C05459=1072.234,347.946,400.424,175.055,31.365,155.656
C05460=1072.241,348.193,400.389,175.059,31.371,155.657
C05461=1072.247,348.441,400.353,175.062,31.376,155.658
C05462=1072.254,348.688,400.318,175.066,31.382,155.659
C05463=1072.260,348.935,400.281,175.070,31.387,155.660
C05464=1072.266,349.183,400.246,175.073,31.392,155.661
C05465=1072.273,349.430,400.210,175.076,31.398,155.663
C05466=1072.279,349.678,400.175,175.080,31.403,155.664
C05467=1072.285,349.925,400.138,175.084,31.409,155.665
C05468=1072.292,350.172,400.103,175.087,31.415,155.666
C05469=1072.298,350.420,400.067,175.091,31.420,155.667
C05470=1072.304,350.667,400.031,175.095,31.426,155.668
C05471=1072.311,350.914,399.996,175.098,31.431,155.669
C05472=1072.317,351.162,399.960,175.101,31.436,155.670
C05473=1072.323,351.409,399.924,175.105,31.442,155.671
C05474=1072.330,351.656,399.889,175.109,31.448,155.672
C05475=1072.336,351.904,399.852,175.112,31.453,155.673
C05476=1072.342,352.151,399.816,175.116,31.458,155.674
C05477=1072.349,352.398,399.780,175.120,31.464,155.675
C05478=1072.356,352.646,399.745,175.123,31.470,155.676
C05479=1072.362,352.893,399.708,175.127,31.475,155.677
C05480=1072.368,353.140,399.673,175.131,31.481,155.679
C05481=1072.374,353.387,399.636,175.134,31.487,155.680
C05482=1072.380,353.635,399.600,175.137,31.492,155.681
C05483=1072.387,353.882,399.564,175.141,31.498,155.682
C05484=1072.393,354.129,399.528,175.145,31.503,155.683
C05485=1072.399,354.377,399.492,175.148,31.509,155.684
C05486=1072.406,354.624,399.456,175.152,31.515,155.685
C05487=1072.412,354.871,399.420,175.156,31.521,155.686
C05488=1072.418,355.118,399.384,175.160,31.526,155.687
C05489=1072.425,355.366,399.347,175.163,31.532,155.689
C05490=1072.432,355.613,399.311,175.167,31.537,155.690
C05491=1072.438,355.860,399.274,175.171,31.543,155.691
C05492=1072.444,356.108,399.238,175.174,31.549,155.692
C05493=1072.450,356.355,399.202,175.178,31.555,155.693
C05494=1072.457,356.602,399.165,175.182,31.561,155.694
C05495=1072.463,356.849,399.129,175.186,31.566,155.695
C05496=1072.470,357.097,399.092,175.189,31.572,155.696
C05497=1072.476,357.344,399.056,175.193,31.578,155.698
C05498=1072.482,357.592,399.020,175.197,31.583,155.699
C05499=1072.488,357.812,398.987,175.199,31.588,155.700
C05500=1072.495,358.032,398.955,175.203,31.594,155.701
C05501=1072.500,358.253,398.923,175.206,31.599,155.702
C05502=1072.506,358.474,398.889,175.210,31.604,155.703
C05503=1072.511,358.695,398.857,175.213,31.609,155.704
C05504=1072.517,358.916,398.824,175.216,31.615,155.705
C05505=1072.524,359.136,398.792,175.220,31.619,155.706
C05506=1072.529,359.357,398.759,175.223,31.625,155.707
C05507=1072.536,359.603,398.722,175.227,31.631,155.708
C05508=1072.542,359.851,398.685,175.230,31.637,155.709
C05509=1072.548,360.098,398.648,175.234,31.642,155.710
C05510=1072.554,360.346,398.612,175.238,31.648,155.711
C05511=1072.561,360.593,398.576,175.241,31.654,155.713
C05512=1072.568,360.840,398.539,175.245,31.660,155.714
C05513=1072.574,361.087,398.502,175.249,31.666,155.715
C05514=1072.580,361.334,398.465,175.253,31.672,155.716
C05515=1072.587,361.582,398.428,175.256,31.678,155.717
C05516=1072.593,361.829,398.391,175.260,31.684,155.719
C05517=1072.600,362.075,398.354,175.264,31.690,155.720
C05518=1072.607,362.323,398.317,175.269,31.696,155.721
C05519=1072.613,362.570,398.281,175.272,31.702,155.722
C05520=1072.619,362.817,398.243,175.276,31.708,155.723
C05521=1072.626,363.065,398.206,175.280,31.714,155.724
C05522=1072.632,363.312,398.170,175.284,31.720,155.726
C05523=1072.639,363.558,398.133,175.287,31.726,155.727
C05524=1072.645,363.806,398.095,175.291,31.732,155.728
C05525=1072.652,364.053,398.058,175.295,31.738,155.729
C05526=1072.659,364.300,398.021,175.299,31.744,155.730
C05527=1072.665,364.547,397.984,175.302,31.750,155.732
C05528=1072.671,364.794,397.947,175.306,31.756,155.733
C05529=1072.678,365.041,397.910,175.310,31.762,155.734
C05530=1072.684,365.289,397.873,175.314,31.769,155.735
C05531=1072.691,365.536,397.835,175.318,31.775,155.737
C05532=1072.697,365.783,397.797,175.322,31.781,155.738
C05533=1072.703,366.030,397.761,175.326,31.788,155.739
C05534=1072.710,366.277,397.723,175.330,31.793,155.740
C05535=1072.717,366.524,397.686,175.333,31.800,155.742
C05536=1072.723,366.771,397.649,175.337,31.806,155.743
C05537=1072.729,367.018,397.611,175.341,31.812,155.744
C05538=1072.736,367.265,397.573,175.345,31.819,155.745
C05539=1072.743,367.512,397.536,175.348,31.824,155.747
C05540=1072.749,367.760,397.498,175.353,31.831,155.748
C05541=1072.755,368.006,397.461,175.357,31.837,155.749
C05542=1072.762,368.254,397.423,175.361,31.844,155.751
C05543=1072.768,368.500,397.386,175.364,31.850,155.752
C05544=1072.775,368.748,397.348,175.368,31.856,155.753
C05545=1072.782,368.994,397.311,175.372,31.862,155.754
C05546=1072.788,369.242,397.272,175.376,31.869,155.756
C05547=1072.794,369.489,397.236,175.380,31.875,155.757
C05548=1072.801,369.736,397.198,175.384,31.882,155.758
C05549=1072.808,369.983,397.161,175.388,31.888,155.759
C05550=1072.814,370.230,397.123,175.392,31.894,155.761
C05551=1072.821,370.477,397.085,175.396,31.900,155.762
C05552=1072.828,370.723,397.047,175.399,31.907,155.763
C05553=1072.834,370.971,397.008,175.404,31.913,155.765
C05554=1072.841,371.217,396.971,175.408,31.920,155.766
C05555=1072.847,371.447,396.936,175.412,31.926,155.767
C05556=1072.854,371.676,396.901,175.415,31.932,155.768
C05557=1072.859,371.904,396.866,175.418,31.938,155.770
C05558=1072.865,372.134,396.830,175.422,31.944,155.771
C05559=1072.872,372.363,396.796,175.426,31.950,155.772
C05560=1072.878,372.592,396.761,175.430,31.956,155.773
C05561=1072.884,372.821,396.725,175.433,31.962,155.774
C05562=1072.890,373.051,396.690,175.437,31.968,155.776
C05563=1072.897,373.297,396.653,175.441,31.974,155.777
C05564=1072.904,373.544,396.614,175.445,31.981,155.778
C05565=1072.910,373.792,396.576,175.450,31.988,155.780
C05566=1072.916,374.038,396.538,175.453,31.994,155.781
C05567=1072.923,374.285,396.499,175.457,32.001,155.782
C05568=1072.929,374.533,396.461,175.461,32.007,155.784
C05569=1072.936,374.778,396.423,175.466,32.014,155.785
C05570=1072.943,375.026,396.385,175.470,32.021,155.787
C05571=1072.950,375.273,396.346,175.473,32.028,155.788
C05572=1072.956,375.520,396.308,175.477,32.034,155.789
C05573=1072.962,375.766,396.269,175.482,32.041,155.791
C05574=1072.969,376.014,396.231,175.486,32.048,155.792
C05575=1072.976,376.260,396.192,175.490,32.054,155.793
C05576=1072.982,376.508,396.154,175.493,32.061,155.795
C05577=1072.988,376.754,396.116,175.498,32.068,155.796
C05578=1072.995,377.001,396.077,175.502,32.075,155.798
C05579=1073.002,377.248,396.040,175.506,32.082,155.799
C05580=1073.009,377.495,396.001,175.511,32.089,155.801
C05581=1073.016,377.742,395.962,175.514,32.095,155.802
C05582=1073.023,377.989,395.924,175.518,32.102,155.803
C05583=1073.029,378.235,395.885,175.523,32.109,155.805
C05584=1073.036,378.482,395.846,175.527,32.116,155.806
C05585=1073.042,378.729,395.808,175.531,32.123,155.808
C05586=1073.049,378.976,395.769,175.534,32.129,155.809
C05587=1073.056,379.223,395.731,175.539,32.136,155.810
C05588=1073.062,379.470,395.692,175.543,32.143,155.812
C05589=1073.069,379.717,395.653,175.547,32.150,155.813
C05590=1073.076,379.964,395.614,175.552,32.157,155.815
C05591=1073.083,380.210,395.575,175.556,32.164,155.816
C05592=1073.090,380.457,395.536,175.560,32.171,155.818
C05593=1073.096,380.703,395.498,175.564,32.178,155.819
C05594=1073.103,380.951,395.459,175.568,32.185,155.820
C05595=1073.110,381.197,395.420,175.573,32.192,155.822
C05596=1073.117,381.445,395.381,175.577,32.199,155.823
C05597=1073.124,381.691,395.342,175.581,32.206,155.825
C05598=1073.131,381.938,395.303,175.585,32.213,155.826
C05599=1073.136,382.185,395.264,175.589,32.220,155.828
C05600=1073.143,382.431,395.225,175.594,32.227,155.829
C05601=1073.150,382.678,395.186,175.598,32.235,155.831
C05602=1073.157,382.924,395.147,175.602,32.241,155.832
C05603=1073.163,383.172,395.108,175.607,32.249,155.834
C05604=1073.170,383.418,395.069,175.610,32.256,155.835
C05605=1073.177,383.665,395.029,175.614,32.263,155.837
C05606=1073.183,383.912,394.990,175.619,32.271,155.838
C05607=1073.190,384.159,394.951,175.623,32.278,155.840
C05608=1073.197,384.405,394.911,175.628,32.285,155.841
C05609=1073.204,384.652,394.873,175.632,32.292,155.843
C05610=1073.211,384.899,394.832,175.637,32.300,155.845
C05611=1073.217,385.142,394.794,175.640,32.307,155.846
C05612=1073.224,385.386,394.755,175.644,32.314,155.848
C05613=1073.231,385.630,394.716,175.649,32.321,155.849
C05614=1073.237,385.873,394.677,175.653,32.328,155.851
C05615=1073.244,386.117,394.638,175.658,32.336,155.852
C05616=1073.250,386.361,394.599,175.662,32.343,155.854
C05617=1073.257,386.605,394.560,175.666,32.350,155.855
C05618=1073.264,386.848,394.521,175.670,32.358,155.857
C05619=1073.270,387.096,394.481,175.674,32.365,155.858
C05620=1073.278,387.342,394.442,175.679,32.373,155.860
C05621=1073.285,387.588,394.402,175.683,32.380,155.862
C05622=1073.291,387.836,394.362,175.688,32.388,155.863
C05623=1073.299,388.082,394.323,175.692,32.395,155.865
C05624=1073.305,388.328,394.283,175.697,32.402,155.866
C05625=1073.312,388.575,394.244,175.701,32.410,155.868
C05626=1073.319,388.822,394.204,175.706,32.418,155.870
C05627=1073.326,389.069,394.164,175.709,32.425,155.871
C05628=1073.333,389.315,394.124,175.714,32.432,155.873
C05629=1073.339,389.561,394.084,175.718,32.440,155.874
C05630=1073.347,389.808,394.044,175.723,32.448,155.876
C05631=1073.354,390.055,394.005,175.728,32.456,155.878
C05632=1073.361,390.301,393.964,175.732,32.463,155.879
C05633=1073.368,390.549,393.925,175.737,32.471,155.881
C05634=1073.374,390.795,393.885,175.741,32.478,155.882
C05635=1073.382,391.042,393.845,175.746,32.486,155.884
C05636=1073.388,391.289,393.805,175.749,32.494,155.886
C05637=1073.396,391.534,393.765,175.754,32.502,155.887
C05638=1073.403,391.781,393.724,175.759,32.509,155.889
C05639=1073.409,392.028,393.684,175.763,32.517,155.891
C05640=1073.416,392.274,393.645,175.768,32.525,155.893
C05641=1073.423,392.521,393.604,175.772,32.533,155.894
C05642=1073.430,392.768,393.564,175.777,32.541,155.896
C05643=1073.437,393.013,393.524,175.782,32.548,155.897
C05644=1073.444,393.261,393.483,175.786,32.556,155.899
C05645=1073.450,393.507,393.443,175.791,32.564,155.901
C05646=1073.457,393.754,393.402,175.795,32.573,155.903
C05647=1073.465,394.000,393.362,175.800,32.580,155.904
C05648=1073.472,394.247,393.322,175.805,32.588,155.906
C05649=1073.478,394.494,393.282,175.808,32.596,155.908
C05650=1073.486,394.740,393.240,175.813,32.604,155.909
C05651=1073.492,394.987,393.200,175.818,32.613,155.911
C05652=1073.500,395.233,393.160,175.822,32.620,155.913
C05653=1073.506,395.480,393.119,175.827,32.628,155.915
C05654=1073.514,395.726,393.078,175.832,32.637,155.917
C05655=1073.520,395.973,393.038,175.836,32.645,155.918
C05656=1073.527,396.219,392.997,175.841,32.653,155.920
C05657=1073.534,396.466,392.957,175.846,32.661,155.922
C05658=1073.541,396.712,392.915,175.850,32.669,155.924
C05659=1073.548,396.959,392.874,175.855,32.678,155.925
C05660=1073.555,397.205,392.835,175.860,32.686,155.927
C05661=1073.563,397.452,392.793,175.864,32.694,155.929
C05662=1073.570,397.698,392.752,175.869,32.702,155.931
C05663=1073.576,397.945,392.712,175.874,32.711,155.933
C05664=1073.584,398.191,392.671,175.878,32.718,155.934
C05665=1073.591,398.438,392.630,175.883,32.727,155.936
C05666=1073.598,398.684,392.589,175.888,32.735,155.938
C05667=1073.605,398.941,392.546,175.893,32.744,155.940
C05668=1073.612,399.197,392.503,175.898,32.753,155.942
C05669=1073.620,399.453,392.460,175.903,32.762,155.944
C05670=1073.627,399.709,392.418,175.908,32.771,155.946
C05671=1073.634,399.956,392.376,175.912,32.779,155.948
C05672=1073.641,400.202,392.335,175.917,32.787,155.949
C05673=1073.648,400.448,392.294,175.922,32.796,155.951
C05674=1073.655,400.695,392.253,175.927,32.805,155.953
C05675=1073.663,400.942,392.212,175.931,32.813,155.955
C05676=1073.669,401.188,392.170,175.936,32.822,155.957
C05677=1073.676,401.434,392.129,175.941,32.830,155.959
C05678=1073.683,401.681,392.088,175.946,32.839,155.961
C05679=1073.690,401.928,392.047,175.951,32.847,155.963
C05680=1073.698,402.174,392.005,175.955,32.856,155.965
C05681=1073.705,402.421,391.964,175.960,32.865,155.966
C05682=1073.712,402.667,391.922,175.965,32.873,155.968
C05683=1073.719,402.914,391.880,175.970,32.882,155.970
C05684=1073.726,403.160,391.839,175.975,32.891,155.972
C05685=1073.733,403.405,391.798,175.980,32.900,155.974
C05686=1073.741,403.652,391.756,175.985,32.909,155.976
C05687=1073.747,403.899,391.715,175.989,32.917,155.978
C05688=1073.755,404.145,391.673,175.994,32.926,155.980
C05689=1073.762,404.392,391.631,175.999,32.935,155.982
C05690=1073.769,404.638,391.589,176.004,32.944,155.984
C05691=1073.776,404.884,391.548,176.009,32.953,155.986
C05692=1073.784,405.130,391.506,176.014,32.962,155.988
C05693=1073.790,405.377,391.464,176.019,32.971,155.990
C05694=1073.798,405.623,391.422,176.024,32.980,155.992
C05695=1073.805,405.870,391.380,176.030,32.989,155.994
C05696=1073.812,406.116,391.338,176.035,32.998,155.996
C05697=1073.819,406.362,391.296,176.039,33.007,155.998
C05698=1073.826,406.609,391.254,176.044,33.016,156.000
C05699=1073.834,406.855,391.212,176.049,33.026,156.002
C05700=1073.841,407.101,391.170,176.054,33.035,156.004
C05701=1073.848,407.348,391.127,176.059,33.044,156.006
C05702=1073.855,407.595,391.086,176.064,33.053,156.008
C05703=1073.862,407.841,391.043,176.069,33.063,156.010
C05704=1073.870,408.087,391.001,176.074,33.072,156.012
C05705=1073.877,408.333,390.959,176.079,33.081,156.015
C05706=1073.884,408.580,390.916,176.085,33.090,156.017
C05707=1073.891,408.826,390.874,176.090,33.100,156.019
C05708=1073.898,409.072,390.832,176.095,33.109,156.021
C05709=1073.906,409.319,390.789,176.100,33.119,156.023
C05710=1073.913,409.565,390.747,176.105,33.128,156.025
C05711=1073.920,409.811,390.704,176.110,33.137,156.027
C05712=1073.928,410.057,390.662,176.116,33.147,156.029
C05713=1073.934,410.303,390.620,176.121,33.157,156.031
C05714=1073.942,410.550,390.577,176.127,33.166,156.034
C05715=1073.950,410.796,390.534,176.132,33.175,156.036
C05716=1073.957,411.042,390.492,176.137,33.185,156.038
C05717=1073.963,411.288,390.449,176.142,33.195,156.040
C05718=1073.972,411.535,390.407,176.147,33.204,156.042
C05719=1073.979,411.781,390.364,176.152,33.214,156.044
C05720=1073.986,412.027,390.321,176.158,33.224,156.047
C05721=1073.993,412.274,390.278,176.164,33.233,156.049
C05722=1074.001,412.519,390.236,176.169,33.243,156.051
C05723=1074.009,412.779,390.190,176.174,33.254,156.053
C05724=1074.017,413.038,390.145,176.180,33.264,156.056
C05725=1074.024,413.298,390.100,176.186,33.274,156.058
C05726=1074.032,413.558,390.055,176.192,33.284,156.060
C05727=1074.040,413.804,390.012,176.197,33.294,156.063
C05728=1074.047,414.050,389.968,176.202,33.304,156.065
C05729=1074.055,414.297,389.925,176.207,33.314,156.067
C05730=1074.063,414.542,389.883,176.213,33.324,156.069
C05731=1074.070,414.789,389.840,176.219,33.334,156.072
C05732=1074.077,415.035,389.797,176.224,33.344,156.074
C05733=1074.085,415.281,389.753,176.229,33.354,156.076
C05734=1074.092,415.527,389.710,176.235,33.364,156.078
C05735=1074.100,415.774,389.667,176.241,33.374,156.081
C05736=1074.107,416.019,389.624,176.246,33.385,156.083
C05737=1074.115,416.266,389.580,176.251,33.395,156.086
C05738=1074.122,416.512,389.537,176.257,33.405,156.088
C05739=1074.129,416.758,389.493,176.263,33.415,156.090
C05740=1074.137,417.004,389.450,176.268,33.425,156.093
C05741=1074.144,417.250,389.406,176.274,33.436,156.095
C05742=1074.152,417.496,389.363,176.280,33.446,156.097
C05743=1074.159,417.742,389.319,176.285,33.456,156.100
C05744=1074.167,417.988,389.276,176.291,33.467,156.102
C05745=1074.174,418.234,389.232,176.296,33.477,156.105
C05746=1074.182,418.480,389.188,176.302,33.488,156.107
C05747=1074.189,418.726,389.144,176.308,33.499,156.109
C05748=1074.197,418.972,389.101,176.313,33.509,156.112
C05749=1074.204,419.218,389.057,176.320,33.519,156.114
C05750=1074.212,419.464,389.013,176.325,33.530,156.117
C05751=1074.220,419.711,388.969,176.330,33.541,156.119
C05752=1074.227,419.956,388.926,176.337,33.551,156.121
C05753=1074.235,420.202,388.881,176.342,33.562,156.124
C05754=1074.243,420.448,388.838,176.348,33.573,156.126
C05755=1074.250,420.694,388.793,176.354,33.583,156.129
C05756=1074.258,420.941,388.749,176.360,33.594,156.131
C05757=1074.266,421.186,388.705,176.365,33.605,156.134
C05758=1074.273,421.432,388.662,176.372,33.615,156.136
C05759=1074.282,421.678,388.617,176.377,33.627,156.139
C05760=1074.289,421.924,388.572,176.383,33.638,156.142
C05761=1074.297,422.170,388.529,176.389,33.648,156.144
C05762=1074.303,422.416,388.484,176.395,33.660,156.147
C05763=1074.311,422.661,388.440,176.401,33.670,156.149
C05764=1074.319,422.907,388.396,176.407,33.682,156.152
C05765=1074.327,423.154,388.351,176.413,33.692,156.154
C05766=1074.335,423.400,388.307,176.419,33.704,156.157
C05767=1074.342,423.646,388.262,176.425,33.715,156.160
C05768=1074.350,423.891,388.218,176.431,33.726,156.162
C05769=1074.358,424.137,388.173,176.437,33.737,156.165
C05770=1074.365,424.383,388.128,176.444,33.748,156.167
C05771=1074.373,424.629,388.084,176.449,33.760,156.170
C05772=1074.381,424.875,388.039,176.456,33.771,156.173
C05773=1074.389,425.121,387.995,176.461,33.783,156.175
C05774=1074.396,425.367,387.950,176.467,33.794,156.178
C05775=1074.405,425.612,387.905,176.474,33.805,156.181
C05776=1074.412,425.858,387.860,176.480,33.817,156.184
C05777=1074.420,426.104,387.816,176.486,33.828,156.186
C05778=1074.427,426.350,387.771,176.492,33.839,156.189
C05779=1074.437,426.627,387.720,176.499,33.853,156.192
C05780=1074.446,426.905,387.669,176.507,33.866,156.195
C05781=1074.455,427.182,387.618,176.513,33.879,156.198
C05782=1074.464,427.459,387.568,176.521,33.892,156.201
C05783=1074.471,427.705,387.523,176.527,33.904,156.204
C05784=1074.479,427.951,387.477,176.533,33.915,156.207
C05785=1074.487,428.197,387.433,176.539,33.928,156.210
C05786=1074.495,428.443,387.387,176.546,33.939,156.212
C05787=1074.503,428.688,387.341,176.552,33.951,156.215
C05788=1074.510,428.934,387.296,176.559,33.963,156.218
C05789=1074.518,429.179,387.251,176.565,33.975,156.221
C05790=1074.527,429.425,387.205,176.571,33.987,156.224
C05791=1074.534,429.671,387.160,176.578,33.999,156.227
C05792=1074.542,429.917,387.115,176.584,34.011,156.230
C05793=1074.551,430.163,387.069,176.591,34.023,156.232
C05794=1074.558,430.408,387.024,176.598,34.035,156.235
C05795=1074.566,430.654,386.978,176.604,34.047,156.238
C05796=1074.574,430.900,386.932,176.611,34.060,156.241
C05797=1074.582,431.145,386.887,176.618,34.072,156.244
C05798=1074.590,431.390,386.841,176.624,34.084,156.247
C05799=1074.598,431.636,386.795,176.630,34.097,156.250
C05800=1074.606,431.882,386.750,176.637,34.109,156.253
C05801=1074.614,432.128,386.704,176.643,34.121,156.256
C05802=1074.622,432.373,386.657,176.650,34.134,156.259
C05803=1074.630,432.619,386.611,176.657,34.146,156.262
C05804=1074.638,432.864,386.566,176.663,34.159,156.265
C05805=1074.646,433.109,386.519,176.670,34.171,156.268
C05806=1074.654,433.355,386.473,176.677,34.184,156.271
C05807=1074.662,433.601,386.428,176.684,34.197,156.274
C05808=1074.670,433.846,386.381,176.690,34.209,156.277
C05809=1074.678,434.092,386.335,176.698,34.223,156.280
C05810=1074.687,434.337,386.289,176.705,34.235,156.283
C05811=1074.694,434.583,386.243,176.712,34.248,156.286
C05812=1074.703,434.828,386.196,176.719,34.261,156.290
C05813=1074.711,435.074,386.149,176.725,34.274,156.293
C05814=1074.719,435.319,386.104,176.732,34.287,156.296
C05815=1074.728,435.565,386.057,176.739,34.300,156.299
C05816=1074.735,435.809,386.011,176.746,34.313,156.302
C05817=1074.743,436.055,385.963,176.754,34.326,156.305
C05818=1074.752,436.301,385.917,176.760,34.339,156.308
C05819=1074.760,436.547,385.871,176.767,34.352,156.312
C05820=1074.768,436.792,385.824,176.774,34.365,156.315
C05821=1074.777,437.037,385.778,176.781,34.378,156.318
C05822=1074.785,437.283,385.731,176.789,34.392,156.321
C05823=1074.794,437.528,385.684,176.796,34.405,156.325
C05824=1074.802,437.773,385.638,176.803,34.418,156.328
C05825=1074.809,438.019,385.590,176.810,34.432,156.331
C05826=1074.818,438.264,385.544,176.818,34.445,156.334
C05827=1074.827,438.509,385.496,176.825,34.459,156.338
C05828=1074.835,438.755,385.449,176.831,34.472,156.341
C05829=1074.844,439.000,385.403,176.839,34.486,156.344
C05830=1074.852,439.246,385.355,176.846,34.499,156.348
C05831=1074.861,439.491,385.308,176.853,34.513,156.351
C05832=1074.869,439.737,385.261,176.861,34.527,156.354
C05833=1074.877,439.981,385.214,176.868,34.541,156.358
C05834=1074.885,440.227,385.167,176.875,34.555,156.361
C05835=1074.895,440.518,385.110,176.885,34.571,156.365
C05836=1074.906,440.809,385.054,176.894,34.588,156.369
C05837=1074.916,441.103,384.997,176.902,34.604,156.374
C05838=1074.926,441.397,384.941,176.911,34.621,156.378
C05839=1074.935,441.690,384.883,176.921,34.638,156.382
C05840=1074.946,441.985,384.826,176.930,34.655,156.386
C05841=1074.954,442.230,384.778,176.937,34.670,156.390
C05842=1074.963,442.475,384.731,176.945,34.684,156.393
C05843=1074.971,442.720,384.683,176.953,34.698,156.397
C05844=1074.980,442.965,384.635,176.961,34.713,156.400
C05845=1074.988,443.211,384.587,176.968,34.727,156.404
C05846=1074.997,443.456,384.539,176.976,34.742,156.408
C05847=1075.006,443.701,384.491,176.984,34.756,156.411
C05848=1075.014,443.946,384.444,176.992,34.771,156.415
C05849=1075.023,444.191,384.395,177.000,34.785,156.418
C05850=1075.032,444.437,384.347,177.007,34.800,156.422
C05851=1075.040,444.682,384.299,177.015,34.815,156.426
C05852=1075.048,444.927,384.251,177.024,34.829,156.429
C05853=1075.057,445.171,384.202,177.031,34.844,156.433
C05854=1075.066,445.417,384.154,177.039,34.859,156.437
C05855=1075.075,445.662,384.106,177.047,34.874,156.441
C05856=1075.083,445.907,384.058,177.056,34.889,156.445
C05857=1075.092,446.152,384.009,177.063,34.904,156.448
C05858=1075.101,446.396,383.961,177.072,34.919,156.452
C05859=1075.110,446.642,383.912,177.080,34.935,156.456
C05860=1075.118,446.887,383.863,177.088,34.950,156.460
C05861=1075.127,447.131,383.815,177.096,34.965,156.464
C05862=1075.136,447.377,383.765,177.103,34.980,156.467
C05863=1075.145,447.622,383.718,177.111,34.995,156.471
C05864=1075.154,447.867,383.669,177.118,35.010,156.475
C05865=1075.162,448.111,383.620,177.124,35.026,156.479
C05866=1075.171,448.355,383.571,177.131,35.041,156.483
C05867=1075.180,448.600,383.523,177.137,35.056,156.487
C05868=1075.190,448.845,383.474,177.144,35.071,156.491
C05869=1075.201,449.089,383.427,177.149,35.085,156.494
C05870=1075.213,449.334,383.380,177.155,35.099,156.498
C05871=1075.226,449.579,383.334,177.161,35.112,156.501
C05872=1075.242,449.825,383.289,177.166,35.124,156.504
C05873=1074.885,449.822,383.050,177.148,35.277,156.545
C05874=1074.870,449.576,383.095,177.141,35.264,156.542
C05875=1074.856,449.331,383.142,177.136,35.251,156.538
C05876=1074.844,449.085,383.188,177.130,35.238,156.535
C05877=1074.832,448.841,383.235,177.124,35.223,156.531
C05878=1074.823,448.596,383.284,177.117,35.209,156.527
C05879=1074.814,448.352,383.333,177.111,35.193,156.523
C05880=1074.805,448.108,383.381,177.104,35.178,156.519
C05881=1074.796,447.863,383.430,177.098,35.163,156.516
C05882=1074.787,447.619,383.478,177.090,35.148,156.512
C05883=1074.778,447.374,383.527,177.083,35.133,156.508
C05884=1074.769,447.129,383.577,177.075,35.118,156.504
C05885=1074.761,446.884,383.625,177.067,35.102,156.500
C05886=1074.752,446.639,383.674,177.059,35.088,156.496
C05887=1074.742,446.394,383.723,177.051,35.072,156.492
C05888=1074.734,446.149,383.771,177.042,35.057,156.489
C05889=1074.725,445.904,383.820,177.034,35.042,156.485
C05890=1074.717,445.659,383.869,177.025,35.027,156.481
C05891=1074.707,445.414,383.916,177.018,35.012,156.477
C05892=1074.699,445.169,383.965,177.010,34.997,156.474
C05893=1074.691,444.924,384.013,177.001,34.982,156.470
C05894=1074.681,444.679,384.062,176.994,34.968,156.466
C05895=1074.673,444.434,384.110,176.985,34.953,156.462
C05896=1074.665,444.189,384.158,176.977,34.938,156.459
C05897=1074.655,443.944,384.206,176.970,34.924,156.455
C05898=1074.647,443.698,384.254,176.962,34.909,156.451
C05899=1074.639,443.453,384.302,176.953,34.895,156.448
C05900=1074.630,443.208,384.350,176.946,34.880,156.444
C05901=1074.622,442.963,384.398,176.938,34.866,156.441
C05902=1074.613,442.717,384.446,176.930,34.851,156.437
C05903=1074.604,442.472,384.494,176.922,34.837,156.433
C05904=1074.596,442.227,384.541,176.915,34.823,156.430
C05905=1074.587,441.982,384.589,176.907,34.808,156.426
C05906=1074.579,441.772,384.631,176.901,34.796,156.423
C05907=1074.573,441.561,384.671,176.894,34.784,156.420
C05908=1074.565,441.349,384.713,176.887,34.772,156.417
C05909=1074.558,441.139,384.753,176.881,34.760,156.414
C05910=1074.551,440.927,384.794,176.874,34.748,156.411
C05911=1074.543,440.717,384.835,176.868,34.736,156.408
C05912=1074.536,440.506,384.877,176.861,34.724,156.405
C05913=1074.529,440.295,384.917,176.855,34.712,156.402
C05914=1074.520,440.050,384.964,176.847,34.698,156.399
C05915=1074.512,439.805,385.012,176.839,34.684,156.395
C05916=1074.503,439.559,385.058,176.832,34.670,156.392
C05917=1074.495,439.314,385.106,176.824,34.657,156.389
C05918=1074.487,439.068,385.153,176.817,34.643,156.385
C05919=1074.478,438.823,385.200,176.809,34.630,156.382
C05920=1074.469,438.578,385.247,176.802,34.616,156.379
C05921=1074.462,438.332,385.295,176.795,34.602,156.375
C05922=1074.453,438.087,385.341,176.788,34.589,156.372
C05923=1074.445,437.842,385.388,176.780,34.576,156.369
C05924=1074.436,437.597,385.435,176.773,34.562,156.365
C05925=1074.428,437.351,385.482,176.766,34.549,156.362
C05926=1074.419,437.106,385.529,176.758,34.536,156.359
C05927=1074.411,436.860,385.575,176.751,34.522,156.356
C05928=1074.403,436.615,385.622,176.744,34.509,156.352
C05929=1074.395,436.370,385.669,176.737,34.496,156.349
C05930=1074.386,436.124,385.716,176.730,34.483,156.346
C05931=1074.378,435.879,385.762,176.722,34.470,156.343
C05932=1074.370,435.633,385.808,176.716,34.457,156.340
C05933=1074.362,435.388,385.855,176.709,34.444,156.337
C05934=1074.353,435.142,385.902,176.702,34.431,156.333
C05935=1074.345,434.898,385.948,176.695,34.418,156.330
C05936=1074.337,434.651,385.994,176.688,34.405,156.327
C05937=1074.329,434.407,386.040,176.681,34.392,156.324
C05938=1074.320,434.161,386.087,176.674,34.380,156.321
C05939=1074.313,433.915,386.134,176.667,34.367,156.318
C05940=1074.305,433.670,386.180,176.660,34.354,156.315
C05941=1074.297,433.424,386.226,176.653,34.341,156.312
C05942=1074.289,433.179,386.272,176.646,34.328,156.309
C05943=1074.280,432.933,386.318,176.639,34.316,156.306
C05944=1074.273,432.687,386.364,176.632,34.304,156.303
C05945=1074.264,432.442,386.411,176.626,34.291,156.299
C05946=1074.257,432.196,386.456,176.619,34.278,156.296
C05947=1074.248,431.950,386.502,176.612,34.266,156.293
C05948=1074.241,431.705,386.548,176.605,34.253,156.290
C05949=1074.232,431.460,386.594,176.600,34.241,156.287
C05950=1074.223,431.192,386.644,176.592,34.228,156.284
C05951=1074.215,430.924,386.694,176.585,34.215,156.281
C05952=1074.206,430.656,386.743,176.577,34.201,156.278
C05953=1074.197,430.389,386.793,176.570,34.188,156.275
C05954=1074.189,430.142,386.839,176.564,34.176,156.272
C05955=1074.181,429.896,386.884,176.557,34.164,156.269
C05956=1074.174,429.651,386.930,176.550,34.151,156.266
C05957=1074.165,429.405,386.975,176.544,34.140,156.263
C05958=1074.157,429.160,387.021,176.537,34.128,156.260
C05959=1074.149,428.914,387.067,176.531,34.116,156.257
C05960=1074.141,428.668,387.113,176.525,34.104,156.255
C05961=1074.133,428.422,387.157,176.518,34.092,156.252
C05962=1074.125,428.177,387.203,176.511,34.080,156.249
C05963=1074.118,427.931,387.247,176.505,34.068,156.246
C05964=1074.110,427.686,387.293,176.499,34.057,156.243
C05965=1074.102,427.440,387.339,176.493,34.045,156.241
C05966=1074.093,427.183,387.386,176.486,34.033,156.238
C05967=1074.085,426.926,387.433,176.479,34.020,156.235
C05968=1074.077,426.669,387.480,176.473,34.009,156.232
C05969=1074.069,426.412,387.527,176.466,33.996,156.229
C05970=1074.061,426.166,387.571,176.460,33.985,156.226
C05971=1074.053,425.920,387.616,176.453,33.973,156.224
C05972=1074.045,425.675,387.661,176.447,33.962,156.221
C05973=1074.037,425.429,387.706,176.441,33.950,156.218
C05974=1074.029,425.183,387.750,176.434,33.939,156.216
C05975=1074.022,424.937,387.795,176.429,33.928,156.213
C05976=1074.014,424.692,387.840,176.422,33.917,156.210
C05977=1074.007,424.446,387.884,176.416,33.905,156.208
C05978=1073.998,424.200,387.930,176.410,33.894,156.205
C05979=1073.990,423.955,387.974,176.404,33.883,156.202
C05980=1073.983,423.709,388.019,176.398,33.872,156.200
C05981=1073.975,423.463,388.063,176.392,33.860,156.197
C05982=1073.968,423.216,388.107,176.385,33.850,156.195
C05983=1073.960,422.971,388.152,176.380,33.838,156.192
C05984=1073.952,422.724,388.197,176.373,33.827,156.189
C05985=1073.944,422.479,388.241,176.368,33.816,156.187
C05986=1073.936,422.233,388.285,176.361,33.805,156.184
C05987=1073.929,421.987,388.330,176.356,33.794,156.182
C05988=1073.921,421.741,388.374,176.349,33.783,156.179
C05989=1073.914,421.496,388.418,176.344,33.772,156.176
C05990=1073.906,421.249,388.463,176.338,33.761,156.174
C05991=1073.899,421.003,388.506,176.332,33.751,156.171
C05992=1073.891,420.757,388.551,176.326,33.740,156.169
C05993=1073.883,420.511,388.594,176.320,33.730,156.166
C05994=1073.875,420.265,388.639,176.314,33.719,156.164
C05995=1073.868,420.019,388.683,176.308,33.708,156.161
C05996=1073.860,419.774,388.727,176.302,33.697,156.159
C05997=1073.852,419.527,388.770,176.297,33.687,156.157
C05998=1073.845,419.281,388.814,176.290,33.676,156.154
C05999=1073.837,419.035,388.858,176.285,33.666,156.152
C06000=1073.829,418.789,388.902,176.280,33.655,156.149
C06001=1073.822,418.543,388.945,176.273,33.645,156.147
C06002=1073.814,418.297,388.989,176.268,33.634,156.144
C06003=1073.806,418.051,389.033,176.262,33.624,156.142
C06004=1073.799,417.805,389.077,176.256,33.613,156.140
C06005=1073.792,417.559,389.121,176.251,33.603,156.137
C06006=1073.785,417.313,389.164,176.244,33.593,156.135
C06007=1073.777,417.067,389.208,176.239,33.582,156.132
C06008=1073.769,416.820,389.251,176.234,33.572,156.130
C06009=1073.762,416.574,389.294,176.228,33.562,156.128
C06010=1073.754,416.328,389.338,176.222,33.551,156.125
C06011=1073.747,416.082,389.381,176.217,33.541,156.123
C06012=1073.739,415.836,389.425,176.212,33.531,156.121
C06013=1073.732,415.590,389.468,176.205,33.521,156.118
C06014=1073.724,415.344,389.512,176.200,33.511,156.116
C06015=1073.717,415.098,389.555,176.195,33.501,156.114
C06016=1073.710,414.851,389.598,176.189,33.491,156.111
C06017=1073.702,414.605,389.642,176.183,33.481,156.109
C06018=1073.694,414.360,389.684,176.178,33.471,156.107
C06019=1073.686,414.113,389.727,176.172,33.461,156.105
C06020=1073.679,413.867,389.770,176.167,33.451,156.102
C06021=1073.672,413.621,389.814,176.161,33.441,156.100
C06022=1073.663,413.360,389.859,176.156,33.431,156.098
C06023=1073.656,413.099,389.905,176.149,33.420,156.095
C06024=1073.648,412.838,389.949,176.144,33.410,156.093
C06025=1073.639,412.577,389.996,176.139,33.399,156.091
C06026=1073.632,412.330,390.039,176.133,33.390,156.088
C06027=1073.625,412.085,390.080,176.127,33.380,156.086
C06028=1073.617,411.838,390.124,176.122,33.370,156.084
C06029=1073.610,411.592,390.167,176.117,33.361,156.082
C06030=1073.603,411.346,390.210,176.112,33.351,156.080
C06031=1073.595,411.100,390.252,176.107,33.341,156.077
C06032=1073.588,410.853,390.295,176.101,33.332,156.075
C06033=1073.581,410.607,390.337,176.096,33.322,156.073
C06034=1073.573,410.361,390.380,176.090,33.313,156.071
C06035=1073.566,410.115,390.423,176.085,33.304,156.069
C06036=1073.559,409.868,390.465,176.080,33.294,156.067
C06037=1073.551,409.622,390.507,176.074,33.284,156.065
C06038=1073.544,409.375,390.550,176.069,33.275,156.062
C06039=1073.537,409.129,390.593,176.064,33.266,156.060
C06040=1073.529,408.883,390.635,176.059,33.256,156.058
C06041=1073.523,408.637,390.677,176.054,33.247,156.056
C06042=1073.515,408.391,390.719,176.048,33.238,156.054
C06043=1073.508,408.145,390.762,176.043,33.228,156.052
C06044=1073.501,407.898,390.805,176.038,33.219,156.050
C06045=1073.493,407.652,390.847,176.033,33.210,156.048
C06046=1073.486,407.405,390.889,176.028,33.200,156.046
C06047=1073.479,407.159,390.931,176.023,33.191,156.043
C06048=1073.472,406.913,390.974,176.018,33.182,156.042
C06049=1073.465,406.666,391.015,176.012,33.173,156.039
C06050=1073.458,406.420,391.057,176.007,33.164,156.037
C06051=1073.450,406.174,391.099,176.002,33.155,156.035
C06052=1073.443,405.928,391.142,175.998,33.146,156.033
C06053=1073.436,405.681,391.183,175.993,33.136,156.031
C06054=1073.429,405.435,391.226,175.988,33.128,156.029
C06055=1073.422,405.188,391.267,175.983,33.119,156.027
C06056=1073.414,404.942,391.309,175.977,33.109,156.025
C06057=1073.407,404.696,391.351,175.972,33.100,156.023
C06058=1073.400,404.450,391.393,175.967,33.092,156.021
C06059=1073.392,404.204,391.435,175.962,33.083,156.019
C06060=1073.386,403.957,391.476,175.957,33.074,156.017
C06061=1073.379,403.710,391.518,175.952,33.065,156.015
C06062=1073.371,403.464,391.560,175.948,33.056,156.013
C06063=1073.364,403.217,391.601,175.943,33.047,156.011
C06064=1073.357,402.971,391.643,175.938,33.038,156.009
C06065=1073.350,402.725,391.685,175.933,33.030,156.008
C06066=1073.342,402.478,391.726,175.928,33.021,156.006
C06067=1073.335,402.231,391.767,175.922,33.012,156.004
C06068=1073.328,401.985,391.810,175.918,33.004,156.002
C06069=1073.321,401.739,391.851,175.913,32.995,156.000
C06070=1073.314,401.492,391.892,175.908,32.987,155.998
C06071=1073.307,401.246,391.933,175.903,32.978,155.996
C06072=1073.300,401.000,391.974,175.898,32.970,155.994
C06073=1073.292,400.753,392.015,175.894,32.961,155.992
C06074=1073.285,400.506,392.057,175.889,32.952,155.990
C06075=1073.278,400.260,392.099,175.884,32.944,155.989
C06076=1073.271,400.013,392.140,175.879,32.935,155.987
C06077=1073.264,399.768,392.181,175.875,32.927,155.985
C06078=1073.256,399.510,392.224,175.870,32.918,155.983
C06079=1073.249,399.251,392.267,175.865,32.909,155.981
C06080=1073.242,398.994,392.310,175.860,32.901,155.979
C06081=1073.234,398.736,392.353,175.855,32.892,155.977
C06082=1073.228,398.490,392.394,175.850,32.883,155.975
C06083=1073.221,398.243,392.435,175.845,32.875,155.973
C06084=1073.214,397.996,392.476,175.841,32.867,155.972
C06085=1073.206,397.750,392.517,175.836,32.858,155.970
C06086=1073.200,397.504,392.558,175.831,32.850,155.968
C06087=1073.193,397.257,392.598,175.827,32.842,155.966
C06088=1073.185,397.010,392.640,175.822,32.834,155.964
C06089=1073.179,396.764,392.680,175.817,32.826,155.963
C06090=1073.171,396.517,392.720,175.813,32.817,155.961
C06091=1073.164,396.271,392.761,175.808,32.809,155.959
C06092=1073.157,396.025,392.802,175.803,32.801,155.957
C06093=1073.150,395.778,392.843,175.799,32.793,155.956
C06094=1073.143,395.532,392.884,175.794,32.785,155.954
C06095=1073.136,395.285,392.924,175.789,32.776,155.952
C06096=1073.130,395.039,392.965,175.785,32.769,155.950
C06097=1073.122,394.792,393.005,175.780,32.761,155.949
C06098=1073.115,394.546,393.046,175.775,32.752,155.947
C06099=1073.108,394.299,393.087,175.771,32.744,155.945
C06100=1073.101,394.053,393.127,175.766,32.736,155.943
C06101=1073.095,393.806,393.168,175.762,32.729,155.942
C06102=1073.087,393.559,393.207,175.757,32.721,155.940
C06103=1073.080,393.313,393.249,175.752,32.713,155.938
C06104=1073.074,393.066,393.289,175.748,32.705,155.937
C06105=1073.066,392.819,393.329,175.743,32.697,155.935
C06106=1073.060,392.573,393.369,175.739,32.689,155.933
C06107=1073.053,392.327,393.410,175.734,32.681,155.931
C06108=1073.046,392.080,393.450,175.729,32.673,155.930
C06109=1073.039,391.833,393.490,175.725,32.666,155.928
C06110=1073.032,391.586,393.530,175.720,32.658,155.926
C06111=1073.025,391.340,393.570,175.716,32.650,155.925
C06112=1073.018,391.094,393.610,175.711,32.642,155.923
C06113=1073.011,390.846,393.651,175.707,32.635,155.921
C06114=1073.004,390.600,393.690,175.702,32.627,155.920
C06115=1072.997,390.354,393.730,175.697,32.619,155.918
C06116=1072.990,390.107,393.770,175.693,32.611,155.916
C06117=1072.983,389.861,393.810,175.688,32.604,155.915
C06118=1072.977,389.614,393.850,175.684,32.597,155.913
C06119=1072.969,389.367,393.890,175.679,32.589,155.912
C06120=1072.963,389.121,393.930,175.675,32.581,155.910
C06121=1072.955,388.874,393.970,175.671,32.574,155.908
C06122=1072.948,388.627,394.009,175.667,32.566,155.907
C06123=1072.941,388.381,394.050,175.662,32.559,155.905
C06124=1072.935,388.134,394.088,175.658,32.551,155.904
C06125=1072.928,387.888,394.129,175.653,32.544,155.902
C06126=1072.920,387.641,394.168,175.649,32.536,155.900
C06127=1072.913,387.395,394.208,175.644,32.529,155.899
C06128=1072.907,387.147,394.247,175.640,32.521,155.897
C06129=1072.900,386.901,394.287,175.635,32.514,155.896
C06130=1072.893,386.656,394.327,175.631,32.506,155.894
C06131=1072.887,386.412,394.365,175.626,32.499,155.892
C06132=1072.880,386.167,394.405,175.622,32.492,155.891
C06133=1072.873,385.923,394.444,175.618,32.485,155.889
C06134=1072.866,385.678,394.483,175.614,32.477,155.888
C06135=1072.859,385.434,394.522,175.610,32.470,155.886
C06136=1072.853,385.190,394.562,175.605,32.463,155.885
C06137=1072.846,384.945,394.600,175.601,32.456,155.883
C06138=1072.839,384.698,394.640,175.597,32.448,155.882
C06139=1072.833,384.451,394.679,175.592,32.441,155.880
C06140=1072.826,384.205,394.719,175.588,32.434,155.879
C06141=1072.819,383.958,394.758,175.583,32.427,155.877
C06142=1072.813,383.711,394.797,175.579,32.419,155.876
C06143=1072.806,383.465,394.837,175.575,32.412,155.874
C06144=1072.799,383.218,394.875,175.571,32.405,155.873
C06145=1072.792,382.971,394.914,175.567,32.398,155.871
C06146=1072.786,382.725,394.954,175.562,32.390,155.869
C06147=1072.779,382.478,394.993,175.558,32.383,155.868
C06148=1072.772,382.231,395.032,175.554,32.376,155.866
C06149=1072.765,381.984,395.071,175.549,32.369,155.865
C06150=1072.759,381.737,395.110,175.545,32.362,155.863
C06151=1072.752,381.490,395.149,175.541,32.355,155.862
C06152=1072.745,381.244,395.189,175.537,32.348,155.861
C06153=1072.738,380.997,395.228,175.533,32.341,155.859
C06154=1072.731,380.750,395.266,175.528,32.334,155.858
C06155=1072.725,380.504,395.305,175.524,32.327,155.856
C06156=1072.718,380.257,395.344,175.520,32.320,155.855
C06157=1072.711,380.010,395.383,175.515,32.313,155.853
C06158=1072.704,379.763,395.422,175.511,32.306,155.852
C06159=1072.698,379.516,395.460,175.508,32.299,155.850
C06160=1072.691,379.269,395.499,175.503,32.292,155.849
C06161=1072.685,379.023,395.537,175.499,32.285,155.847
C06162=1072.678,378.776,395.576,175.495,32.278,155.846
C06163=1072.671,378.529,395.615,175.490,32.271,155.845
C06164=1072.664,378.282,395.654,175.486,32.264,155.843
C06165=1072.657,378.035,395.693,175.482,32.258,155.842
C06166=1072.651,377.788,395.731,175.479,32.251,155.840
C06167=1072.644,377.541,395.770,175.474,32.244,155.839
C06168=1072.637,377.294,395.808,175.470,32.237,155.838
C06169=1072.631,377.048,395.846,175.466,32.231,155.836
C06170=1072.624,376.801,395.884,175.461,32.223,155.835
C06171=1072.617,376.554,395.923,175.457,32.217,155.833
C06172=1072.611,376.307,395.961,175.453,32.210,155.832
C06173=1072.604,376.060,396.000,175.450,32.203,155.831
C06174=1072.598,375.814,396.039,175.445,32.197,155.829
C06175=1072.591,375.566,396.077,175.441,32.190,155.828
C06176=1072.584,375.320,396.116,175.437,32.183,155.826
C06177=1072.578,375.072,396.154,175.433,32.177,155.825
C06178=1072.571,374.826,396.192,175.428,32.170,155.824
C06179=1072.564,374.579,396.230,175.425,32.163,155.822
C06180=1072.557,374.332,396.269,175.421,32.157,155.821
C06181=1072.552,374.085,396.306,175.417,32.150,155.820
C06182=1072.545,373.838,396.345,175.413,32.143,155.818
C06183=1072.538,373.591,396.383,175.408,32.137,155.817
C06184=1072.532,373.344,396.421,175.404,32.130,155.815
C06185=1072.525,373.097,396.460,175.401,32.124,155.814
C06186=1072.519,372.867,396.495,175.397,32.118,155.813
C06187=1072.512,372.638,396.530,175.393,32.111,155.812
C06188=1072.506,372.408,396.565,175.389,32.105,155.810
C06189=1072.500,372.179,396.601,175.385,32.100,155.809
C06190=1072.493,371.948,396.636,175.381,32.093,155.808
C06191=1072.487,371.719,396.672,175.378,32.087,155.807
C06192=1072.481,371.488,396.706,175.375,32.082,155.806
C06193=1072.475,371.259,396.741,175.371,32.075,155.804
C06194=1072.469,371.012,396.780,175.366,32.069,155.803
C06195=1072.462,370.765,396.817,175.362,32.062,155.802
C06196=1072.455,370.518,396.855,175.359,32.056,155.800
C06197=1072.448,370.271,396.893,175.355,32.050,155.799
C06198=1072.442,370.024,396.931,175.351,32.043,155.798
C06199=1072.436,369.777,396.969,175.347,32.037,155.796
C06200=1072.429,369.530,397.006,175.342,32.031,155.795
C06201=1072.423,369.283,397.044,175.339,32.025,155.794
C06202=1072.415,369.036,397.082,175.335,32.018,155.793
C06203=1072.409,368.789,397.119,175.331,32.012,155.791
C06204=1072.402,368.542,397.157,175.327,32.005,155.790
C06205=1072.396,368.295,397.195,175.323,31.999,155.789
C06206=1072.389,368.047,397.232,175.320,31.993,155.787
C06207=1072.383,367.801,397.269,175.316,31.987,155.786
C06208=1072.376,367.553,397.307,175.311,31.980,155.785
C06209=1072.370,367.307,397.345,175.307,31.974,155.784
C06210=1072.363,367.060,397.382,175.303,31.968,155.782
C06211=1072.357,366.812,397.419,175.300,31.962,155.781
C06212=1072.350,366.565,397.457,175.296,31.956,155.780
C06213=1072.344,366.318,397.494,175.292,31.949,155.779
C06214=1072.337,366.071,397.532,175.288,31.943,155.777
C06215=1072.331,365.824,397.569,175.284,31.937,155.776
C06216=1072.325,365.577,397.606,175.281,31.931,155.775
C06217=1072.318,365.330,397.644,175.277,31.925,155.774
C06218=1072.312,365.083,397.681,175.273,31.918,155.772
C06219=1072.305,364.835,397.719,175.268,31.912,155.771
C06220=1072.299,364.588,397.755,175.264,31.906,155.770
C06221=1072.293,364.342,397.792,175.261,31.900,155.769
C06222=1072.286,364.094,397.830,175.257,31.894,155.767
C06223=1072.280,363.847,397.867,175.253,31.888,155.766
C06224=1072.273,363.600,397.904,175.249,31.882,155.765
C06225=1072.266,363.353,397.941,175.246,31.876,155.764
C06226=1072.260,363.105,397.978,175.242,31.869,155.763
C06227=1072.253,362.859,398.016,175.238,31.864,155.761
C06228=1072.247,362.612,398.052,175.234,31.858,155.760
C06229=1072.240,362.364,398.089,175.230,31.852,155.759
C06230=1072.233,362.117,398.126,175.227,31.846,155.758
C06231=1072.228,361.870,398.163,175.223,31.840,155.757
C06232=1072.221,361.622,398.200,175.219,31.834,155.755
C06233=1072.214,361.376,398.237,175.215,31.828,155.754
C06234=1072.208,361.129,398.273,175.212,31.822,155.753
C06235=1072.201,360.881,398.310,175.208,31.816,155.752
C06236=1072.195,360.634,398.347,175.204,31.810,155.751
C06237=1072.189,360.387,398.384,175.200,31.804,155.750
C06238=1072.182,360.140,398.421,175.196,31.798,155.748
C06239=1072.175,359.893,398.458,175.193,31.792,155.747
C06240=1072.169,359.645,398.494,175.189,31.786,155.746
C06241=1072.163,359.398,398.531,175.185,31.780,155.745
C06242=1072.157,359.178,398.564,175.181,31.775,155.744
C06243=1072.152,358.956,398.597,175.179,31.770,155.743
C06244=1072.146,358.734,398.629,175.175,31.765,155.742
C06245=1072.139,358.513,398.663,175.171,31.760,155.741
C06246=1072.133,358.291,398.695,175.168,31.754,155.740
C06247=1072.128,358.070,398.728,175.164,31.749,155.739
C06248=1072.122,357.848,398.760,175.162,31.744,155.738
C06249=1072.116,357.627,398.793,175.158,31.739,155.737
C06250=1072.110,357.380,398.830,175.154,31.733,155.735
C06251=1072.104,357.133,398.866,175.150,31.728,155.734
C06252=1072.097,356.885,398.902,175.147,31.722,155.733
C06253=1072.090,356.638,398.939,175.143,31.716,155.732
C06254=1072.084,356.391,398.975,175.139,31.710,155.731
C06255=1072.078,356.144,399.012,175.135,31.704,155.730
C06256=1072.071,355.897,399.048,175.132,31.698,155.729
C06257=1072.065,355.649,399.085,175.129,31.693,155.728
C06258=1072.059,355.402,399.120,175.125,31.687,155.726
C06259=1072.052,355.154,399.157,175.121,31.681,155.725
C06260=1072.045,354.907,399.193,175.118,31.676,155.724
C06261=1072.039,354.660,399.229,175.114,31.670,155.723
C06262=1072.033,354.413,399.265,175.110,31.665,155.722
C06263=1072.026,354.166,399.302,175.106,31.659,155.721
C06264=1072.020,353.918,399.338,175.103,31.653,155.720
C06265=1072.014,353.671,399.374,175.099,31.647,155.719
C06266=1072.008,353.424,399.410,175.095,31.642,155.718
C06267=1072.001,353.177,399.447,175.091,31.636,155.716
C06268=1071.995,352.929,399.482,175.088,31.631,155.715
C06269=1071.988,352.682,399.518,175.085,31.625,155.714
C06270=1071.982,352.435,399.554,175.081,31.619,155.713
C06271=1071.976,352.188,399.590,175.077,31.614,155.712
C06272=1071.970,351.940,399.626,175.074,31.609,155.711
C06273=1071.962,351.692,399.662,175.070,31.603,155.710
C06274=1071.956,351.445,399.698,175.066,31.597,155.709
C06275=1071.950,351.198,399.735,175.062,31.592,155.708
C06276=1071.944,350.950,399.770,175.059,31.586,155.707
C06277=1071.937,350.703,399.805,175.056,31.581,155.706
C06278=1071.930,350.456,399.842,175.052,31.575,155.705
C06279=1071.924,350.208,399.878,175.049,31.570,155.703
C06280=1071.918,349.961,399.913,175.045,31.564,155.702
C06281=1071.911,349.713,399.949,175.041,31.559,155.701
C06282=1071.905,349.466,399.985,175.037,31.553,155.700
C06283=1071.899,349.218,400.020,175.034,31.548,155.699
C06284=1071.892,348.971,400.056,175.031,31.543,155.698
C06285=1071.886,348.725,400.091,175.027,31.537,155.697
C06286=1071.880,348.477,400.127,175.023,31.532,155.696
C06287=1071.874,348.229,400.163,175.020,31.526,155.695
C06288=1071.867,347.982,400.198,175.016,31.521,155.694
C06289=1071.861,347.735,400.234,175.012,31.515,155.693
C06290=1071.855,347.487,400.270,175.009,31.510,155.692
C06291=1071.848,347.240,400.305,175.006,31.505,155.691
C06292=1071.842,346.992,400.341,175.002,31.499,155.690
C06293=1071.835,346.745,400.376,174.998,31.494,155.689
C06294=1071.829,346.497,400.412,174.995,31.489,155.688
C06295=1071.823,346.251,400.446,174.991,31.483,155.687
C06296=1071.817,346.003,400.482,174.988,31.478,155.686
C06297=1071.810,345.756,400.517,174.984,31.472,155.685
C06298=1071.805,345.536,400.549,174.982,31.468,155.684
C06299=1071.799,345.317,400.580,174.978,31.463,155.683
C06300=1071.794,345.096,400.612,174.975,31.458,155.682
C06301=1071.788,344.877,400.644,174.971,31.454,155.681
C06302=1071.783,344.657,400.675,174.969,31.449,155.680
C06303=1071.777,344.437,400.706,174.966,31.444,155.679
C06304=1071.771,344.219,400.737,174.962,31.439,155.678
C06305=1071.766,343.999,400.768,174.959,31.434,155.677
C06306=1071.760,343.751,400.804,174.956,31.430,155.676
C06307=1071.753,343.504,400.839,174.952,31.424,155.675
C06308=1071.746,343.256,400.874,174.949,31.419,155.674
C06309=1071.741,343.009,400.909,174.946,31.414,155.673
C06310=1071.734,342.762,400.944,174.942,31.408,155.672
C06311=1071.728,342.514,400.979,174.938,31.404,155.672
C06312=1071.721,342.266,401.014,174.935,31.398,155.670
C06313=1071.715,342.018,401.049,174.932,31.393,155.669
C06314=1071.709,341.772,401.084,174.928,31.388,155.668
C06315=1071.702,341.524,401.119,174.924,31.382,155.667
C06316=1071.696,341.276,401.154,174.922,31.378,155.667
C06317=1071.690,341.030,401.189,174.918,31.372,155.665
C06318=1071.684,340.782,401.224,174.914,31.367,155.665
C06319=1071.677,340.534,401.259,174.911,31.362,155.664
C06320=1071.671,340.286,401.294,174.908,31.357,155.663
C06321=1071.665,340.039,401.328,174.904,31.352,155.662
C06322=1071.658,339.792,401.364,174.900,31.347,155.661
C06323=1071.652,339.544,401.398,174.898,31.341,155.660
C06324=1071.646,339.297,401.433,174.894,31.336,155.659
C06325=1071.640,339.049,401.468,174.890,31.331,155.658
C06326=1071.633,338.802,401.503,174.887,31.326,155.657
C06327=1071.627,338.554,401.537,174.884,31.321,155.656
C06328=1071.621,338.307,401.573,174.880,31.316,155.655
C06329=1071.615,338.059,401.607,174.876,31.311,155.654
C06330=1071.609,337.811,401.641,174.874,31.305,155.653
C06331=1071.602,337.564,401.676,174.870,31.301,155.652
C06332=1071.596,337.317,401.710,174.866,31.296,155.651
C06333=1071.590,337.069,401.745,174.863,31.290,155.650
C06334=1071.583,336.821,401.780,174.860,31.285,155.649
C06335=1071.577,336.574,401.814,174.856,31.280,155.648
C06336=1071.571,336.326,401.848,174.853,31.276,155.647
C06337=1071.564,336.079,401.884,174.850,31.270,155.646
C06338=1071.558,335.831,401.918,174.846,31.265,155.645
C06339=1071.552,335.583,401.952,174.843,31.260,155.644
C06340=1071.546,335.336,401.986,174.840,31.255,155.643
C06341=1071.539,335.088,402.020,174.836,31.250,155.643
C06342=1071.533,334.841,402.055,174.833,31.246,155.642
C06343=1071.527,334.593,402.090,174.829,31.240,155.641
C06344=1071.521,334.346,402.124,174.826,31.235,155.640
C06345=1071.514,334.098,402.158,174.823,31.230,155.639
C06346=1071.508,333.850,402.193,174.819,31.226,155.638
C06347=1071.502,333.603,402.227,174.816,31.221,155.637
C06348=1071.496,333.355,402.261,174.813,31.216,155.636
C06349=1071.490,333.108,402.295,174.809,31.211,155.635
C06350=1071.484,332.860,402.329,174.807,31.206,155.634
C06351=1071.477,332.612,402.364,174.803,31.201,155.633
C06352=1071.472,332.365,402.398,174.799,31.196,155.632
C06353=1071.465,332.117,402.432,174.797,31.191,155.631
C06354=1071.459,331.895,402.463,174.794,31.187,155.630
C06355=1071.454,331.673,402.494,174.790,31.182,155.630
C06356=1071.449,331.451,402.524,174.787,31.178,155.629
C06357=1071.443,331.229,402.554,174.785,31.173,155.628
C06358=1071.437,331.007,402.585,174.782,31.169,155.627
C06359=1071.431,330.785,402.616,174.778,31.164,155.626
C06360=1071.425,330.562,402.646,174.775,31.160,155.626
C06361=1071.420,330.341,402.676,174.773,31.156,155.625
C06362=1071.414,330.093,402.711,174.769,31.151,155.624
C06363=1071.408,329.845,402.744,174.766,31.147,155.623
C06364=1071.401,329.597,402.778,174.763,31.142,155.622
C06365=1071.395,329.350,402.812,174.759,31.137,155.621
C06366=1071.388,329.102,402.846,174.756,31.132,155.620
C06367=1071.382,328.854,402.879,174.753,31.127,155.620
C06368=1071.376,328.607,402.913,174.750,31.123,155.619
C06369=1071.369,328.359,402.947,174.746,31.118,155.618
C06370=1071.364,328.111,402.980,174.743,31.113,155.617
C06371=1071.356,327.864,403.014,174.740,31.108,155.616
C06372=1071.351,327.616,403.048,174.736,31.103,155.615
C06373=1071.344,327.368,403.082,174.733,31.099,155.614
C06374=1071.338,327.121,403.115,174.730,31.094,155.613
C06375=1071.332,326.874,403.150,174.727,31.089,155.612
C06376=1071.325,326.625,403.183,174.723,31.085,155.612
C06377=1071.319,326.378,403.217,174.721,31.080,155.611
C06378=1071.313,326.130,403.249,174.717,31.075,155.610
C06379=1071.306,325.882,403.284,174.713,31.071,155.609
C06380=1071.300,325.635,403.317,174.711,31.066,155.608
C06381=1071.294,325.388,403.351,174.707,31.061,155.607
C06382=1071.288,325.139,403.384,174.704,31.057,155.606
C06383=1071.282,324.892,403.418,174.701,31.052,155.606
C06384=1071.276,324.644,403.451,174.698,31.047,155.605
C06385=1071.269,324.397,403.485,174.694,31.042,155.604
C06386=1071.263,324.148,403.518,174.692,31.037,155.603
C06387=1071.257,323.901,403.551,174.688,31.033,155.602
C06388=1071.251,323.654,403.585,174.685,31.028,155.601
C06389=1071.245,323.406,403.618,174.682,31.023,155.600
C06390=1071.239,323.157,403.652,174.679,31.019,155.600
C06391=1071.232,322.910,403.685,174.675,31.014,155.599
C06392=1071.227,322.663,403.718,174.672,31.010,155.598
C06393=1071.220,322.415,403.751,174.669,31.005,155.597
C06394=1071.214,322.168,403.785,174.666,31.000,155.596
C06395=1071.207,321.919,403.818,174.662,30.995,155.595
C06396=1071.202,321.671,403.852,174.660,30.991,155.594
C06397=1071.196,321.424,403.884,174.656,30.986,155.594
C06398=1071.189,321.177,403.918,174.653,30.981,155.593
C06399=1071.183,320.929,403.951,174.650,30.977,155.592
C06400=1071.177,320.681,403.984,174.647,30.972,155.591
C06401=1071.171,320.433,404.018,174.643,30.967,155.590
C06402=1071.165,320.185,404.050,174.641,30.963,155.589
C06403=1071.159,319.937,404.084,174.637,30.958,155.588
C06404=1071.153,319.690,404.117,174.634,30.953,155.588
C06405=1071.147,319.442,404.150,174.631,30.949,155.587
C06406=1071.141,319.195,404.183,174.628,30.944,155.586
C06407=1071.134,318.947,404.216,174.625,30.940,155.585
C06408=1071.129,318.699,404.249,174.622,30.935,155.584
C06409=1071.123,318.452,404.282,174.619,30.930,155.583
C06410=1071.117,318.226,404.312,174.616,30.926,155.583
C06411=1071.112,318.002,404.342,174.613,30.922,155.582
C06412=1071.106,317.775,404.372,174.610,30.918,155.581
C06413=1071.101,317.550,404.402,174.607,30.914,155.580
C06414=1071.096,317.325,404.432,174.605,30.909,155.580
C06415=1071.090,317.100,404.463,174.602,30.905,155.579
C06416=1071.085,316.875,404.492,174.599,30.901,155.578
C06417=1071.079,316.649,404.522,174.596,30.897,155.577
C06418=1071.073,316.402,404.555,174.593,30.892,155.576
C06419=1071.067,316.154,404.588,174.590,30.888,155.576
C06420=1071.061,315.906,404.621,174.586,30.883,155.575
C06421=1071.055,315.658,404.654,174.584,30.878,155.574
C06422=1071.049,315.411,404.686,174.581,30.874,155.573
C06423=1071.043,315.162,404.719,174.577,30.870,155.572
C06424=1071.038,314.915,404.751,174.575,30.865,155.571
C06425=1071.031,314.668,404.784,174.571,30.860,155.571
C06426=1071.026,314.420,404.818,174.568,30.855,155.570
C06427=1071.019,314.172,404.850,174.566,30.851,155.569
C06428=1071.013,313.924,404.882,174.562,30.847,155.568
C06429=1071.007,313.677,404.915,174.559,30.842,155.567
C06430=1071.000,313.429,404.948,174.556,30.838,155.567
C06431=1070.994,313.180,404.980,174.553,30.833,155.566
C06432=1070.987,312.933,405.012,174.550,30.829,155.565
C06433=1070.981,312.685,405.044,174.547,30.825,155.564
C06434=1070.975,312.437,405.077,174.544,30.820,155.563
C06435=1070.969,312.189,405.110,174.540,30.816,155.563
C06436=1070.963,311.942,405.141,174.538,30.811,155.562
C06437=1070.957,311.694,405.174,174.535,30.807,155.561
C06438=1070.951,311.446,405.206,174.531,30.803,155.560
C06439=1070.944,311.199,405.238,174.529,30.798,155.559
C06440=1070.938,310.951,405.270,174.525,30.794,155.559
C06441=1070.932,310.703,405.303,174.522,30.790,155.558
C06442=1070.926,310.455,405.335,174.520,30.785,155.557
C06443=1070.919,310.207,405.368,174.516,30.781,155.556
C06444=1070.913,309.959,405.400,174.513,30.776,155.556
C06445=1070.907,309.711,405.433,174.510,30.772,155.555
C06446=1070.900,309.463,405.464,174.507,30.768,155.554
C06447=1070.894,309.216,405.497,174.504,30.763,155.553
C06448=1070.889,308.968,405.529,174.501,30.759,155.552
C06449=1070.883,308.720,405.561,174.498,30.754,155.552
C06450=1070.876,308.472,405.593,174.496,30.750,155.551
C06451=1070.870,308.225,405.625,174.492,30.746,155.550
C06452=1070.864,307.976,405.657,174.489,30.741,155.549
C06453=1070.857,307.729,405.690,174.487,30.737,155.548
C06454=1070.852,307.481,405.721,174.483,30.732,155.548
C06455=1070.846,307.233,405.753,174.480,30.728,155.547
C06456=1070.839,306.986,405.785,174.477,30.724,155.546
C06457=1070.833,306.738,405.817,174.474,30.719,155.545
C06458=1070.828,306.490,405.849,174.471,30.715,155.545
C06459=1070.822,306.242,405.881,174.468,30.710,155.544
C06460=1070.815,305.994,405.914,174.465,30.706,155.543
C06461=1070.809,305.746,405.945,174.462,30.702,155.542
C06462=1070.803,305.499,405.977,174.459,30.697,155.541
C06463=1070.797,305.251,406.009,174.456,30.693,155.541
C06464=1070.791,305.002,406.041,174.453,30.689,155.540
C06465=1070.784,304.755,406.073,174.450,30.684,155.539
C06466=1070.780,304.532,406.101,174.447,30.680,155.538
C06467=1070.775,304.308,406.130,174.445,30.677,155.538
C06468=1070.769,304.084,406.158,174.443,30.673,155.537
C06469=1070.763,303.861,406.187,174.440,30.669,155.536
C06470=1070.757,303.637,406.216,174.437,30.665,155.536
C06471=1070.752,303.414,406.245,174.435,30.661,155.535
C06472=1070.747,303.190,406.274,174.432,30.657,155.534
C06473=1070.742,302.967,406.302,174.429,30.653,155.534
C06474=1070.736,302.719,406.334,174.426,30.649,155.533
C06475=1070.730,302.471,406.366,174.423,30.644,155.532
C06476=1070.723,302.224,406.397,174.420,30.640,155.531
C06477=1070.717,301.975,406.429,174.417,30.636,155.530
C06478=1070.711,301.727,406.461,174.414,30.631,155.530
C06479=1070.705,301.480,406.492,174.411,30.627,155.529
C06480=1070.699,301.232,406.524,174.409,30.623,155.528
C06481=1070.694,300.984,406.556,174.405,30.618,155.527
C06482=1070.688,300.736,406.588,174.402,30.614,155.527
C06483=1070.682,300.488,406.618,174.400,30.610,155.526
C06484=1070.676,300.240,406.650,174.397,30.606,155.525
C06485=1070.671,299.993,406.682,174.394,30.601,155.524
C06486=1070.664,299.745,406.713,174.391,30.597,155.524
C06487=1070.658,299.496,406.745,174.388,30.592,155.523
C06488=1070.653,299.249,406.777,174.386,30.588,155.522
C06489=1070.646,299.000,406.808,174.382,30.583,155.521
C06490=1070.641,298.753,406.839,174.379,30.579,155.520
C06491=1070.634,298.505,406.871,174.377,30.575,155.520
C06492=1070.629,298.257,406.903,174.374,30.571,155.519
C06493=1070.623,298.009,406.934,174.370,30.566,155.518
C06494=1070.617,297.761,406.965,174.368,30.562,155.517
C06495=1070.611,297.513,406.997,174.365,30.558,155.517
C06496=1070.605,297.266,407.028,174.363,30.553,155.516
C06497=1070.599,297.017,407.059,174.359,30.549,155.515
C06498=1070.593,296.770,407.090,174.356,30.545,155.514
C06499=1070.587,296.521,407.122,174.354,30.541,155.514
C06500=1070.581,296.274,407.153,174.351,30.537,155.513
C06501=1070.575,296.026,407.184,174.347,30.532,155.512
C06502=1070.569,295.778,407.215,174.345,30.528,155.511
C06503=1070.563,295.530,407.247,174.342,30.524,155.511
C06504=1070.557,295.282,407.277,174.339,30.520,155.510
C06505=1070.551,295.034,407.309,174.337,30.515,155.509
C06506=1070.545,294.786,407.339,174.333,30.511,155.509
C06507=1070.538,294.538,407.371,174.330,30.507,155.508
C06508=1070.533,294.290,407.402,174.328,30.503,155.507
C06509=1070.527,294.042,407.433,174.325,30.499,155.506
C06510=1070.521,293.794,407.463,174.322,30.494,155.506
C06511=1070.514,293.546,407.494,174.319,30.490,155.505
C06512=1070.509,293.298,407.526,174.316,30.486,155.504
C06513=1070.503,293.050,407.557,174.314,30.482,155.503
C06514=1070.496,292.803,407.588,174.311,30.478,155.503
C06515=1070.491,292.555,407.618,174.307,30.473,155.502
C06516=1070.485,292.306,407.649,174.305,30.469,155.501
C06517=1070.479,292.059,407.680,174.302,30.465,155.500
C06518=1070.472,291.810,407.711,174.299,30.461,155.500
C06519=1070.467,291.562,407.741,174.297,30.457,155.499
C06520=1070.460,291.315,407.773,174.294,30.453,155.498
C06521=1070.455,291.066,407.804,174.291,30.449,155.498
C06522=1070.449,290.850,407.830,174.289,30.445,155.497
C06523=1070.444,290.634,407.857,174.286,30.441,155.496
C06524=1070.440,290.418,407.884,174.284,30.437,155.496
C06525=1070.434,290.202,407.910,174.281,30.434,155.495
C06526=1070.428,289.986,407.938,174.279,30.430,155.494
C06527=1070.423,289.770,407.964,174.277,30.426,155.494
C06528=1070.418,289.554,407.991,174.274,30.423,155.493
C06529=1070.413,289.338,408.018,174.271,30.419,155.492
C06530=1070.406,289.089,408.048,174.269,30.415,155.492
C06531=1070.401,288.841,408.079,174.266,30.411,155.491
C06532=1070.395,288.593,408.109,174.263,30.407,155.490
C06533=1070.388,288.345,408.140,174.261,30.403,155.490
C06534=1070.382,288.098,408.171,174.257,30.398,155.489
C06535=1070.376,287.850,408.201,174.254,30.395,155.488
C06536=1070.370,287.601,408.232,174.252,30.391,155.488
C06537=1070.364,287.354,408.262,174.249,30.386,155.487
C06538=1070.358,287.105,408.293,174.246,30.382,155.486
C06539=1070.352,286.857,408.323,174.244,30.378,155.485
C06540=1070.346,286.609,408.354,174.241,30.374,155.485
C06541=1070.340,286.362,408.384,174.238,30.370,155.484
C06542=1070.334,286.113,408.415,174.235,30.366,155.483
C06543=1070.328,285.865,408.445,174.232,30.361,155.482
C06544=1070.323,285.617,408.475,174.230,30.358,155.482
C06545=1070.316,285.368,408.505,174.227,30.353,155.481
C06546=1070.310,285.120,408.536,174.224,30.349,155.480
C06547=1070.305,284.873,408.566,174.222,30.346,155.480
C06548=1070.299,284.625,408.596,174.219,30.341,155.479
C06549=1070.292,284.377,408.627,174.216,30.337,155.478
C06550=1070.286,284.129,408.657,174.213,30.333,155.477
C06551=1070.280,283.881,408.687,174.210,30.329,155.477
C06552=1070.274,283.632,408.717,174.208,30.325,155.476
C06553=1070.268,283.384,408.748,174.205,30.321,155.475
C06554=1070.262,283.136,408.778,174.203,30.316,155.475
C06555=1070.256,282.888,408.808,174.200,30.312,155.474
C06556=1070.251,282.640,408.839,174.197,30.308,155.473
C06557=1070.245,282.392,408.868,174.195,30.304,155.472
C06558=1070.239,282.144,408.899,174.192,30.300,155.472
C06559=1070.232,281.896,408.929,174.188,30.296,155.471
C06560=1070.227,281.648,408.958,174.186,30.292,155.470
C06561=1070.221,281.400,408.989,174.183,30.288,155.470
C06562=1070.215,281.152,409.019,174.181,30.284,155.469
C06563=1070.209,280.903,409.049,174.178,30.279,155.468
C06564=1070.203,280.655,409.079,174.175,30.275,155.468
C06565=1070.197,280.407,409.110,174.173,30.271,155.467
C06566=1070.191,280.159,409.139,174.170,30.267,155.466
C06567=1070.185,279.911,409.169,174.167,30.263,155.465
C06568=1070.180,279.663,409.199,174.165,30.259,155.465
C06569=1070.172,279.415,409.229,174.162,30.255,155.464
C06570=1070.167,279.167,409.259,174.160,30.251,155.463
C06571=1070.161,278.918,409.289,174.156,30.247,155.463
C06572=1070.155,278.671,409.319,174.153,30.243,155.462
C06573=1070.149,278.422,409.348,174.151,30.239,155.461
C06574=1070.143,278.174,409.379,174.148,30.234,155.461
C06575=1070.137,277.926,409.408,174.146,30.231,155.460
C06576=1070.131,277.678,409.437,174.143,30.227,155.459
C06577=1070.125,277.429,409.468,174.140,30.222,155.458
C06578=1070.120,277.219,409.493,174.139,30.219,155.458
C06579=1070.114,277.007,409.518,174.136,30.216,155.457
C06580=1070.109,276.797,409.543,174.133,30.212,155.457
C06581=1070.104,276.586,409.569,174.132,30.209,155.456
C06582=1070.100,276.375,409.594,174.129,30.205,155.455
C06583=1070.094,276.163,409.619,174.127,30.202,155.455
C06584=1070.089,275.953,409.645,174.125,30.199,155.454
C06585=1070.084,275.741,409.670,174.122,30.195,155.454
C06586=1070.078,275.493,409.699,174.119,30.191,155.453
C06587=1070.072,275.245,409.729,174.117,30.187,155.452
C06588=1070.067,274.997,409.759,174.114,30.183,155.452
C06589=1070.060,274.749,409.788,174.112,30.179,155.451
C06590=1070.055,274.500,409.818,174.109,30.175,155.450
C06591=1070.049,274.252,409.847,174.106,30.171,155.450
C06592=1070.043,274.004,409.877,174.104,30.167,155.449
C06593=1070.037,273.756,409.906,174.101,30.163,155.448
C06594=1070.031,273.508,409.936,174.099,30.158,155.447
C06595=1070.025,273.260,409.965,174.096,30.154,155.447
C06596=1070.019,273.012,409.995,174.093,30.151,155.446
C06597=1070.013,272.764,410.024,174.091,30.146,155.445
C06598=1070.007,272.515,410.054,174.088,30.142,155.445
C06599=1070.001,272.267,410.083,174.085,30.138,155.444
C06600=1069.995,272.019,410.112,174.083,30.135,155.443
C06601=1069.989,271.771,410.142,174.080,30.130,155.443
C06602=1069.983,271.523,410.171,174.078,30.126,155.442
C06603=1069.977,271.274,410.200,174.075,30.122,155.441
C06604=1069.971,271.026,410.229,174.072,30.119,155.441
C06605=1069.965,270.778,410.258,174.070,30.114,155.440
C06606=1069.959,270.530,410.289,174.067,30.110,155.439
C06607=1069.953,270.282,410.318,174.065,30.106,155.439
C06608=1069.947,270.033,410.347,174.062,30.103,155.438
C06609=1069.941,269.785,410.377,174.059,30.098,155.437
C06610=1069.935,269.537,410.406,174.057,30.094,155.436
C06611=1069.930,269.288,410.434,174.054,30.090,155.436
C06612=1069.923,269.040,410.464,174.052,30.086,155.435
C06613=1069.917,268.792,410.493,174.049,30.082,155.434
C06614=1069.912,268.544,410.522,174.046,30.078,155.434
C06615=1069.906,268.296,410.551,174.044,30.074,155.433
C06616=1069.900,268.048,410.580,174.041,30.070,155.432
C06617=1069.893,267.800,410.609,174.039,30.066,155.432
C06618=1069.888,267.551,410.639,174.036,30.062,155.431
C06619=1069.882,267.303,410.668,174.033,30.058,155.430
C06620=1069.876,267.054,410.696,174.031,30.054,155.430
C06621=1069.870,266.806,410.725,174.028,30.050,155.429
C06622=1069.863,266.558,410.754,174.026,30.046,155.428
C06623=1069.858,266.310,410.784,174.023,30.042,155.428
C06624=1069.852,266.062,410.813,174.021,30.038,155.427
C06625=1069.846,265.814,410.841,174.019,30.035,155.426
C06626=1069.840,265.565,410.870,174.016,30.030,155.426
C06627=1069.834,265.317,410.899,174.014,30.026,155.425
C06628=1069.828,265.069,410.928,174.011,30.022,155.424
C06629=1069.822,264.820,410.957,174.008,30.018,155.424
C06630=1069.816,264.572,410.986,174.006,30.014,155.423
C06631=1069.810,264.325,411.014,174.003,30.010,155.422
C06632=1069.804,264.076,411.043,174.001,30.006,155.421
C06633=1069.799,263.827,411.072,173.998,30.002,155.421
C06634=1069.788,263.409,411.121,173.994,29.995,155.420
C06635=1069.778,262.990,411.169,173.990,29.989,155.419
C06636=1069.768,262.571,411.217,173.985,29.982,155.417
C06637=1069.758,262.153,411.265,173.981,29.976,155.416
C06638=1069.752,261.905,411.294,173.978,29.972,155.416
C06639=1069.746,261.656,411.323,173.976,29.968,155.415
C06640=1069.739,261.408,411.352,173.973,29.964,155.414
C06641=1069.733,261.160,411.379,173.971,29.960,155.414
C06642=1069.726,260.911,411.408,173.969,29.956,155.413
C06643=1069.721,260.663,411.436,173.966,29.952,155.412
C06644=1069.715,260.415,411.465,173.964,29.948,155.412
C06645=1069.709,260.166,411.494,173.961,29.944,155.411
C06646=1069.703,259.918,411.522,173.959,29.940,155.410
C06647=1069.697,259.670,411.551,173.956,29.937,155.410
C06648=1069.691,259.422,411.579,173.953,29.933,155.409
C06649=1069.684,259.174,411.607,173.951,29.929,155.408
C06650=1069.678,258.925,411.636,173.948,29.924,155.408
C06651=1069.672,258.676,411.664,173.946,29.920,155.407
C06652=1069.667,258.429,411.693,173.943,29.917,155.406
C06653=1069.661,258.180,411.721,173.941,29.913,155.406
C06654=1069.655,257.931,411.749,173.939,29.909,155.405
C06655=1069.648,257.683,411.778,173.936,29.905,155.404
C06656=1069.643,257.435,411.806,173.934,29.901,155.404
C06657=1069.637,257.187,411.834,173.931,29.897,155.403
C06658=1069.631,256.938,411.863,173.929,29.893,155.402
C06659=1069.624,256.690,411.892,173.926,29.889,155.402
C06660=1069.618,256.442,411.919,173.923,29.885,155.401
C06661=1069.612,256.193,411.947,173.921,29.881,155.400
C06662=1069.607,255.945,411.976,173.919,29.877,155.400
C06663=1069.601,255.697,412.004,173.917,29.873,155.399
C06664=1069.595,255.448,412.033,173.914,29.870,155.398
C06665=1069.588,255.200,412.060,173.912,29.865,155.398
C06666=1069.583,254.952,412.088,173.909,29.861,155.397
C06667=1069.577,254.703,412.117,173.906,29.857,155.396
C06668=1069.571,254.454,412.145,173.904,29.853,155.396
C06669=1069.566,254.206,412.173,173.902,29.850,155.395
C06670=1069.559,253.958,412.201,173.900,29.846,155.394
C06671=1069.553,253.710,412.229,173.897,29.841,155.394
C06672=1069.547,253.462,412.258,173.894,29.837,155.393
C06673=1069.541,253.213,412.286,173.892,29.833,155.392
C06674=1069.535,252.965,412.313,173.889,29.830,155.392
C06675=1069.529,252.716,412.342,173.887,29.826,155.391
C06676=1069.524,252.468,412.370,173.885,29.822,155.390
C06677=1069.518,252.220,412.398,173.883,29.817,155.390
C06678=1069.511,251.971,412.426,173.880,29.814,155.389
C06679=1069.506,251.723,412.454,173.877,29.810,155.388
C06680=1069.500,251.474,412.482,173.875,29.806,155.388
C06681=1069.495,251.226,412.510,173.872,29.802,155.387
C06682=1069.488,250.978,412.538,173.871,29.798,155.386
C06683=1069.483,250.730,412.566,173.868,29.794,155.386
C06684=1069.477,250.481,412.594,173.866,29.790,155.385
C06685=1069.471,250.233,412.621,173.863,29.786,155.384
C06686=1069.463,249.907,412.658,173.860,29.781,155.383
C06687=1069.456,249.582,412.694,173.857,29.775,155.382
C06688=1069.448,249.256,412.731,173.854,29.770,155.381
C06689=1069.441,248.932,412.768,173.850,29.765,155.381
C06690=1069.431,248.549,412.810,173.847,29.758,155.380
C06691=1069.426,248.301,412.838,173.845,29.754,155.379
C06692=1069.420,248.052,412.866,173.842,29.750,155.378
C06693=1069.415,247.803,412.893,173.840,29.747,155.378
C06694=1069.408,247.555,412.921,173.838,29.742,155.377
C06695=1069.403,247.307,412.949,173.835,29.738,155.376
C06696=1069.397,247.058,412.978,173.833,29.734,155.376
C06697=1069.391,246.810,413.004,173.831,29.731,155.375
C06698=1069.386,246.561,413.032,173.829,29.726,155.374
C06699=1069.379,246.313,413.060,173.826,29.722,155.373
C06700=1069.374,246.064,413.087,173.823,29.718,155.373
C06701=1069.367,245.816,413.115,173.821,29.714,155.372
C06702=1069.362,245.568,413.143,173.819,29.711,155.371
C06703=1069.356,245.319,413.170,173.817,29.707,155.371
C06704=1069.350,245.071,413.198,173.814,29.702,155.370
C06705=1069.344,244.822,413.225,173.812,29.698,155.369
C06706=1069.338,244.574,413.252,173.809,29.694,155.369
C06707=1069.333,244.326,413.280,173.808,29.691,155.368
C06708=1069.326,244.077,413.307,173.805,29.687,155.367
C06709=1069.321,243.829,413.335,173.802,29.683,155.367
C06710=1069.315,243.580,413.362,173.800,29.678,155.366
C06711=1069.309,243.332,413.390,173.798,29.675,155.365
C06712=1069.303,243.084,413.417,173.796,29.671,155.365
C06713=1069.297,242.835,413.445,173.793,29.667,155.364
C06714=1069.291,242.587,413.472,173.791,29.663,155.363
C06715=1069.285,242.338,413.499,173.788,29.658,155.363
C06716=1069.279,242.089,413.526,173.787,29.655,155.362
C06717=1069.273,241.841,413.554,173.784,29.651,155.361
C06718=1069.268,241.592,413.581,173.782,29.647,155.361
C06719=1069.261,241.345,413.608,173.779,29.643,155.360
C06720=1069.255,241.096,413.635,173.777,29.639,155.359
C06721=1069.250,240.847,413.663,173.775,29.635,155.359
C06722=1069.243,240.598,413.690,173.772,29.631,155.358
C06723=1069.238,240.350,413.717,173.770,29.627,155.357
C06724=1069.231,240.102,413.744,173.768,29.623,155.357
C06725=1069.226,239.853,413.772,173.766,29.619,155.356
C06726=1069.220,239.605,413.799,173.763,29.615,155.355
C06727=1069.214,239.357,413.826,173.761,29.611,155.355
C06728=1069.208,239.108,413.853,173.759,29.607,155.354
C06729=1069.202,238.859,413.880,173.756,29.603,155.353
C06730=1069.197,238.611,413.907,173.754,29.600,155.353
C06731=1069.190,238.362,413.935,173.751,29.596,155.352
C06732=1069.184,238.114,413.961,173.750,29.591,155.351
C06733=1069.179,237.866,413.988,173.747,29.587,155.351
C06734=1069.172,237.617,414.015,173.745,29.583,155.350
C06735=1069.166,237.369,414.042,173.743,29.580,155.349
C06736=1069.160,237.120,414.069,173.741,29.576,155.349
C06737=1069.155,236.871,414.097,173.738,29.572,155.348
C06738=1069.149,236.623,414.123,173.736,29.567,155.347
C06739=1069.143,236.409,414.146,173.734,29.564,155.347
C06740=1069.139,236.195,414.169,173.732,29.561,155.346
C06741=1069.133,235.982,414.192,173.730,29.558,155.346
C06742=1069.129,235.768,414.216,173.728,29.554,155.345
C06743=1069.123,235.554,414.239,173.727,29.551,155.345
C06744=1069.118,235.340,414.262,173.724,29.547,155.344
C06745=1069.113,235.127,414.285,173.722,29.543,155.343
C06746=1069.108,234.913,414.308,173.721,29.540,155.343
C06747=1069.103,234.665,414.335,173.718,29.536,155.342
C06748=1069.097,234.416,414.362,173.716,29.532,155.342
C06749=1069.091,234.167,414.389,173.714,29.528,155.341
C06750=1069.085,233.919,414.415,173.712,29.524,155.340
C06751=1069.079,233.670,414.442,173.709,29.520,155.339
C06752=1069.073,233.422,414.469,173.708,29.516,155.339
C06753=1069.067,233.173,414.496,173.705,29.513,155.338
C06754=1069.061,232.925,414.522,173.702,29.508,155.337
C06755=1069.055,232.676,414.549,173.701,29.504,155.337
C06756=1069.050,232.428,414.575,173.698,29.500,155.336
C06757=1069.044,232.180,414.602,173.696,29.496,155.335
C06758=1069.037,231.931,414.629,173.693,29.492,155.335
C06759=1069.032,231.682,414.656,173.692,29.489,155.334
C06760=1069.026,231.434,414.682,173.689,29.484,155.333
C06761=1069.020,231.185,414.709,173.687,29.480,155.333
C06762=1069.014,230.937,414.736,173.685,29.476,155.332
C06763=1069.009,230.689,414.762,173.683,29.473,155.331
C06764=1069.002,230.440,414.789,173.680,29.469,155.331
C06765=1068.997,230.191,414.815,173.679,29.464,155.330
C06766=1068.991,229.942,414.842,173.676,29.460,155.329
C06767=1068.985,229.694,414.869,173.674,29.456,155.329
C06768=1068.979,229.446,414.895,173.672,29.453,155.328
C06769=1068.973,229.198,414.921,173.670,29.449,155.327
C06770=1068.967,228.948,414.948,173.667,29.445,155.327
C06771=1068.961,228.700,414.974,173.665,29.441,155.326
C06772=1068.955,228.451,415.000,173.663,29.436,155.325
C06773=1068.949,228.203,415.027,173.660,29.432,155.325
C06774=1068.943,227.954,415.053,173.659,29.429,155.324
C06775=1068.937,227.706,415.080,173.656,29.425,155.323
C06776=1068.930,227.457,415.106,173.654,29.421,155.323
C06777=1068.925,227.208,415.132,173.652,29.417,155.322
C06778=1068.919,226.960,415.159,173.650,29.413,155.321
C06779=1068.913,226.711,415.185,173.648,29.409,155.321
C06780=1068.907,226.463,415.211,173.646,29.405,155.320
C06781=1068.901,226.214,415.237,173.643,29.401,155.319
C06782=1068.896,225.966,415.264,173.642,29.397,155.319
C06783=1068.890,225.717,415.290,173.639,29.393,155.318
C06784=1068.884,225.469,415.316,173.637,29.389,155.317
C06785=1068.878,225.221,415.342,173.635,29.385,155.317
C06786=1068.872,224.972,415.368,173.633,29.381,155.316
C06787=1068.866,224.724,415.394,173.630,29.377,155.315
C06788=1068.860,224.474,415.421,173.629,29.373,155.315
C06789=1068.854,224.225,415.447,173.626,29.369,155.314
C06790=1068.848,223.977,415.473,173.625,29.365,155.313
C06791=1068.842,223.728,415.499,173.622,29.361,155.313
C06792=1068.837,223.479,415.525,173.620,29.357,155.312
C06793=1068.831,223.231,415.552,173.618,29.353,155.311
C06794=1068.825,222.982,415.577,173.616,29.349,155.311
C06795=1068.820,222.765,415.601,173.614,29.345,155.310
C06796=1068.814,222.547,415.623,173.612,29.342,155.309
C06797=1068.810,222.329,415.646,173.610,29.338,155.309
C06798=1068.804,222.112,415.668,173.608,29.334,155.308
C06799=1068.799,221.894,415.692,173.607,29.331,155.308
C06800=1068.795,221.676,415.715,173.604,29.327,155.307
C06801=1068.789,221.458,415.737,173.603,29.324,155.306
C06802=1068.784,221.240,415.760,173.601,29.321,155.306
C06803=1068.778,220.992,415.786,173.599,29.316,155.305
C06804=1068.772,220.743,415.812,173.597,29.313,155.304
C06805=1068.766,220.495,415.837,173.594,29.309,155.304
C06806=1068.760,220.247,415.863,173.592,29.305,155.303
C06807=1068.754,219.998,415.889,173.590,29.301,155.303
C06808=1068.748,219.749,415.915,173.588,29.297,155.302
C06809=1068.742,219.501,415.941,173.586,29.293,155.301
C06810=1068.736,219.252,415.967,173.584,29.289,155.300
C06811=1068.731,219.003,415.993,173.581,29.285,155.300
C06812=1068.724,218.754,416.018,173.580,29.281,155.299
C06813=1068.719,218.506,416.045,173.577,29.277,155.299
C06814=1068.712,218.257,416.070,173.576,29.273,155.298
C06815=1068.706,218.009,416.095,173.573,29.269,155.297
C06816=1068.701,217.760,416.121,173.572,29.265,155.296
C06817=1068.694,217.512,416.147,173.569,29.261,155.296
C06818=1068.689,217.263,416.173,173.567,29.256,155.295
C06819=1068.683,217.014,416.199,173.565,29.253,155.294
C06820=1068.677,216.765,416.224,173.563,29.249,155.294
C06821=1068.671,216.516,416.250,173.561,29.245,155.293
C06822=1068.665,216.268,416.275,173.559,29.241,155.292
C06823=1068.659,216.020,416.301,173.557,29.236,155.292
C06824=1068.653,215.771,416.327,173.555,29.233,155.291
C06825=1068.648,215.522,416.353,173.552,29.229,155.290
C06826=1068.642,215.274,416.378,173.551,29.224,155.290
C06827=1068.635,215.025,416.403,173.548,29.220,155.289
C06828=1068.630,214.776,416.429,173.547,29.216,155.288
C06829=1068.624,214.527,416.455,173.544,29.212,155.288
C06830=1068.618,214.279,416.480,173.543,29.208,155.287
C06831=1068.613,214.030,416.506,173.541,29.204,155.286
C06832=1068.606,213.782,416.531,173.539,29.200,155.286
C06833=1068.601,213.533,416.557,173.537,29.196,155.285
C06834=1068.595,213.284,416.582,173.534,29.192,155.284
C06835=1068.589,213.036,416.607,173.533,29.188,155.284
C06836=1068.584,212.787,416.633,173.530,29.184,155.283
C06837=1068.577,212.538,416.658,173.529,29.180,155.282
C06838=1068.571,212.290,416.684,173.526,29.176,155.282
C06839=1068.565,212.041,416.709,173.525,29.172,155.281
C06840=1068.559,211.792,416.734,173.522,29.167,155.280
C06841=1068.554,211.544,416.760,173.521,29.164,155.279
C06842=1068.548,211.295,416.785,173.518,29.160,155.279
C06843=1068.542,211.047,416.811,173.517,29.156,155.278
C06844=1068.535,210.798,416.836,173.514,29.151,155.277
C06845=1068.529,210.549,416.861,173.513,29.148,155.277
C06846=1068.524,210.301,416.887,173.510,29.144,155.276
C06847=1068.518,210.052,416.912,173.508,29.139,155.275
C06848=1068.512,209.803,416.937,173.506,29.135,155.275
C06849=1068.506,209.555,416.962,173.504,29.131,155.274
C06850=1068.500,209.306,416.988,173.502,29.127,155.273
C06851=1068.495,209.091,417.009,173.501,29.124,155.273
C06852=1068.490,208.875,417.031,173.499,29.120,155.272
C06853=1068.485,208.660,417.053,173.497,29.116,155.272
C06854=1068.480,208.445,417.075,173.495,29.113,155.271
C06855=1068.474,208.229,417.097,173.494,29.109,155.270
C06856=1068.470,208.013,417.119,173.492,29.106,155.270
C06857=1068.465,207.797,417.140,173.491,29.102,155.269
C06858=1068.459,207.582,417.161,173.488,29.099,155.269
C06859=1068.435,206.538,417.264,173.343,29.025,155.265
C06860=1068.429,206.289,417.288,173.341,29.023,155.265
C06861=1068.424,206.041,417.313,173.339,29.019,155.264
C06862=1068.418,205.791,417.337,173.336,29.016,155.264
C06863=1068.412,205.543,417.361,173.335,29.013,155.263
C06864=1068.407,205.294,417.386,173.332,29.010,155.263
C06865=1068.400,205.045,417.410,173.330,29.007,155.262
C06866=1068.395,204.796,417.434,173.328,29.003,155.262
C06867=1068.389,204.548,417.459,173.325,29.001,155.261
C06868=1068.384,204.299,417.484,173.323,28.997,155.261
C06869=1068.378,204.051,417.508,173.321,28.994,155.260
C06870=1068.372,203.802,417.532,173.319,28.991,155.260
C06871=1068.366,203.553,417.556,173.317,28.988,155.259
C06872=1068.361,203.304,417.580,173.314,28.985,155.259
C06873=1068.355,203.055,417.605,173.312,28.981,155.258
C06874=1068.349,202.807,417.629,173.310,28.979,155.258
C06875=1068.344,202.558,417.652,173.308,28.975,155.258
C06876=1068.338,202.308,417.677,173.306,28.972,155.257
C06877=1068.332,202.060,417.700,173.304,28.969,155.257
C06878=1068.327,201.812,417.725,173.301,28.966,155.256
C06879=1068.320,201.563,417.749,173.299,28.963,155.256
C06880=1068.315,201.314,417.773,173.297,28.960,155.255
C06881=1068.308,201.065,417.797,173.294,28.957,155.255
C06882=1068.303,200.816,417.821,173.293,28.954,155.254
C06883=1068.297,200.568,417.845,173.290,28.951,155.254
C06884=1068.291,200.318,417.869,173.289,28.948,155.253
C06885=1068.285,200.070,417.893,173.286,28.945,155.253
C06886=1068.280,199.821,417.917,173.283,28.942,155.253
C06887=1068.273,199.572,417.941,173.282,28.938,155.252
C06888=1068.268,199.324,417.965,173.279,28.936,155.252
C06889=1068.262,199.075,417.988,173.278,28.932,155.251
C06890=1068.256,198.826,418.013,173.275,28.929,155.251
C06891=1068.250,198.577,418.036,173.273,28.927,155.250
C06892=1068.245,198.329,418.061,173.271,28.923,155.250
C06893=1068.239,198.079,418.084,173.268,28.920,155.250
C06894=1068.234,197.831,418.108,173.267,28.918,155.249
C06895=1068.227,197.582,418.132,173.264,28.914,155.249
C06896=1068.221,197.334,418.155,173.262,28.911,155.248
C06897=1068.216,197.084,418.179,173.260,28.908,155.248
C06898=1068.210,196.836,418.203,173.258,28.905,155.247
C06899=1068.205,196.587,418.227,173.256,28.902,155.247
C06900=1068.198,196.338,418.251,173.253,28.899,155.246
C06901=1068.193,196.089,418.275,173.252,28.896,155.246
C06902=1068.187,195.841,418.298,173.249,28.893,155.245
C06903=1068.181,195.592,418.321,173.247,28.890,155.245
C06904=1068.176,195.343,418.346,173.245,28.887,155.245
C06905=1068.169,195.094,418.369,173.243,28.884,155.244
C06906=1068.164,194.845,418.393,173.241,28.881,155.244
C06907=1068.158,194.597,418.417,173.239,28.878,155.243
C06908=1068.153,194.348,418.440,173.237,28.875,155.243
C06909=1068.147,194.099,418.464,173.234,28.872,155.242
C06910=1068.141,193.850,418.487,173.232,28.869,155.242
C06911=1068.135,193.601,418.512,173.230,28.866,155.241
C06912=1068.130,193.352,418.535,173.228,28.863,155.241
C06913=1068.124,193.104,418.559,173.226,28.859,155.241
C06914=1068.119,192.855,418.582,173.224,28.857,155.240
C06915=1068.112,192.606,418.606,173.221,28.854,155.240
C06916=1068.107,192.357,418.629,173.220,28.851,155.239
C06917=1068.101,192.108,418.653,173.217,28.848,155.239
C06918=1068.095,191.859,418.676,173.216,28.844,155.238
C06919=1068.090,191.611,418.700,173.213,28.841,155.238
C06920=1068.083,191.328,418.727,173.211,28.838,155.237
C06921=1068.077,191.047,418.753,173.208,28.834,155.237
C06922=1068.071,190.763,418.780,173.207,28.831,155.236
C06923=1068.065,190.481,418.806,173.204,28.828,155.236
C06924=1068.058,190.232,418.830,173.202,28.825,155.235
C06925=1068.053,189.983,418.854,173.200,28.822,155.235
C06926=1068.047,189.735,418.878,173.197,28.819,155.235
C06927=1068.041,189.486,418.901,173.196,28.816,155.234
C06928=1068.036,189.237,418.924,173.193,28.812,155.234
C06929=1068.030,188.989,418.948,173.192,28.810,155.233
C06930=1068.025,188.740,418.971,173.189,28.807,155.233
C06931=1068.020,188.490,418.994,173.188,28.803,155.232
C06932=1068.013,188.242,419.018,173.185,28.801,155.232
C06933=1068.008,187.993,419.041,173.183,28.797,155.231
C06934=1068.003,187.744,419.064,173.181,28.794,155.231
C06935=1067.997,187.495,419.087,173.179,28.792,155.231
C06936=1067.991,187.247,419.111,173.177,28.788,155.230
C06937=1067.986,186.998,419.135,173.175,28.785,155.230
C06938=1067.980,186.749,419.157,173.173,28.783,155.229
C06939=1067.975,186.500,419.180,173.171,28.779,155.229
C06940=1067.969,186.252,419.204,173.169,28.777,155.228
C06941=1067.964,186.002,419.228,173.167,28.773,155.228
C06942=1067.958,185.753,419.251,173.165,28.770,155.227
C06943=1067.952,185.505,419.274,173.163,28.767,155.227
C06944=1067.947,185.255,419.297,173.161,28.764,155.226
C06945=1067.941,185.007,419.321,173.158,28.761,155.226
C06946=1067.935,184.758,419.344,173.157,28.759,155.226
C06947=1067.930,184.509,419.367,173.154,28.755,155.225
C06948=1067.923,184.260,419.390,173.153,28.752,155.225
C06949=1067.918,184.011,419.413,173.150,28.749,155.224
C06950=1067.912,183.762,419.436,173.149,28.747,155.224
C06951=1067.906,183.513,419.459,173.147,28.744,155.224
C06952=1067.900,183.264,419.482,173.144,28.741,155.223
C06953=1067.894,183.016,419.504,173.143,28.738,155.223
C06954=1067.888,182.767,419.527,173.140,28.735,155.222
C06955=1067.882,182.518,419.550,173.139,28.733,155.222
C06956=1067.877,182.269,419.573,173.136,28.729,155.221
C06957=1067.871,182.020,419.596,173.134,28.726,155.221
C06958=1067.865,181.772,419.620,173.132,28.724,155.221
C06959=1067.859,181.522,419.642,173.130,28.721,155.220
C06960=1067.853,181.274,419.664,173.128,28.718,155.220
C06961=1067.847,181.025,419.687,173.126,28.715,155.219
C06962=1067.842,180.776,419.710,173.124,28.712,155.219
C06963=1067.836,180.527,419.733,173.122,28.709,155.219
C06964=1067.830,180.278,419.756,173.120,28.707,155.218
C06965=1067.824,180.029,419.778,173.118,28.703,155.218
C06966=1067.818,179.781,419.801,173.116,28.701,155.217
C06967=1067.812,179.532,419.824,173.114,28.698,155.217
C06968=1067.806,179.283,419.847,173.112,28.695,155.217
C06969=1067.801,179.034,419.870,173.110,28.692,155.216
C06970=1067.795,178.785,419.893,173.108,28.689,155.216
C06971=1067.788,178.536,419.915,173.106,28.687,155.215
C06972=1067.783,178.287,419.938,173.104,28.684,155.215
C06973=1067.777,178.038,419.960,173.102,28.681,155.215
C06974=1067.772,177.789,419.983,173.100,28.678,155.214
C06975=1067.766,177.540,420.006,173.098,28.675,155.214
C06976=1067.759,177.292,420.029,173.096,28.672,155.213
C06977=1067.754,177.043,420.052,173.094,28.669,155.213
C06978=1067.748,176.793,420.074,173.092,28.666,155.212
C06979=1067.743,176.544,420.097,173.091,28.664,155.212
C06980=1067.736,176.296,420.119,173.088,28.661,155.212
C06981=1067.730,176.047,420.142,173.086,28.658,155.211
C06982=1067.725,175.798,420.165,173.084,28.654,155.211
C06983=1067.719,175.548,420.187,173.082,28.652,155.210
C06984=1067.712,175.266,420.212,173.080,28.649,155.210
C06985=1067.706,174.983,420.238,173.078,28.645,155.209
C06986=1067.700,174.701,420.264,173.076,28.642,155.209
C06987=1067.692,174.418,420.290,173.073,28.639,155.208
C06988=1067.687,174.169,420.312,173.072,28.636,155.208
C06989=1067.681,173.920,420.335,173.069,28.633,155.208
C06990=1067.676,173.671,420.357,173.067,28.630,155.207
C06991=1067.670,173.423,420.380,173.066,28.627,155.207
C06992=1067.664,173.173,420.402,173.063,28.624,155.206
C06993=1067.659,172.924,420.425,173.062,28.622,155.206
C06994=1067.653,172.675,420.448,173.060,28.619,155.206
C06995=1067.647,172.426,420.469,173.058,28.615,155.205
C06996=1067.642,172.178,420.492,173.056,28.613,155.205
C06997=1067.636,171.929,420.515,173.053,28.610,155.204
C06998=1067.630,171.680,420.537,173.052,28.607,155.204
C06999=1067.624,171.431,420.559,173.050,28.604,155.203
C07000=1067.619,171.182,420.582,173.048,28.601,155.203
C07001=1067.613,170.933,420.604,173.046,28.599,155.203
C07002=1067.607,170.684,420.626,173.044,28.595,155.202
C07003=1067.601,170.435,420.649,173.042,28.592,155.202
C07004=1067.596,170.186,420.672,173.040,28.590,155.201
C07005=1067.590,169.937,420.693,173.039,28.587,155.201
C07006=1067.584,169.689,420.716,173.036,28.584,155.201
C07007=1067.579,169.439,420.738,173.035,28.581,155.200
C07008=1067.573,169.191,420.761,173.033,28.578,155.200
C07009=1067.567,168.941,420.783,173.030,28.575,155.199
C07010=1067.562,168.693,420.805,173.029,28.572,155.199
C07011=1067.557,168.444,420.828,173.027,28.570,155.198
C07012=1067.550,168.194,420.849,173.025,28.567,155.198
C07013=1067.545,167.945,420.872,173.023,28.564,155.198
C07014=1067.540,167.697,420.894,173.022,28.561,155.197
C07015=1067.533,167.448,420.916,173.019,28.558,155.197
C07016=1067.528,167.199,420.939,173.017,28.555,155.196
C07017=1067.523,166.950,420.961,173.016,28.552,155.196
C07018=1067.517,166.701,420.983,173.013,28.549,155.195
C07019=1067.511,166.452,421.005,173.012,28.546,155.195
C07020=1067.505,166.204,421.027,173.010,28.543,155.195
C07021=1067.500,165.954,421.049,173.008,28.540,155.194
C07022=1067.495,165.705,421.072,173.006,28.538,155.194
C07023=1067.489,165.457,421.094,173.004,28.535,155.193
C07024=1067.483,165.207,421.116,173.003,28.532,155.193
C07025=1067.478,164.958,421.139,173.000,28.529,155.192
C07026=1067.472,164.710,421.160,172.999,28.526,155.192
C07027=1067.467,164.460,421.182,172.997,28.523,155.192
C07028=1067.461,164.211,421.204,172.995,28.520,155.191
C07029=1067.455,163.963,421.226,172.993,28.517,155.191
C07030=1067.450,163.714,421.249,172.991,28.514,155.190
C07031=1067.444,163.464,421.270,172.989,28.511,155.190
C07032=1067.439,163.216,421.293,172.987,28.508,155.189
C07033=1067.433,162.967,421.315,172.986,28.506,155.189
C07034=1067.428,162.718,421.336,172.984,28.503,155.189
C07035=1067.422,162.469,421.359,172.982,28.499,155.188
C07036=1067.416,162.220,421.381,172.980,28.497,155.188
C07037=1067.411,161.971,421.403,172.978,28.494,155.187
C07038=1067.405,161.722,421.425,172.976,28.491,155.187
C07039=1067.400,161.473,421.446,172.974,28.488,155.187
C07040=1067.394,161.224,421.469,172.973,28.485,155.186
C07041=1067.388,160.974,421.490,172.971,28.482,155.186
C07042=1067.382,160.727,421.512,172.969,28.479,155.185
C07043=1067.377,160.477,421.534,172.967,28.477,155.185
C07044=1067.371,160.228,421.556,172.965,28.474,155.184
C07045=1067.365,159.979,421.577,172.964,28.471,155.184
C07046=1067.360,159.730,421.600,172.961,28.468,155.184
C07047=1067.354,159.481,421.621,172.960,28.465,155.183
C07048=1067.347,159.198,421.646,172.957,28.462,155.183
C07049=1067.340,158.914,421.670,172.956,28.459,155.182
C07050=1067.335,158.631,421.695,172.953,28.456,155.182
C07051=1067.327,158.348,421.720,172.952,28.453,155.181
C07052=1067.322,158.099,421.741,172.949,28.450,155.181
C07053=1067.316,157.850,421.763,172.947,28.447,155.181
C07054=1067.311,157.601,421.785,172.946,28.444,155.180
C07055=1067.305,157.352,421.806,172.944,28.442,155.180
C07056=1067.299,157.103,421.828,172.942,28.439,155.179
C07057=1067.293,156.855,421.849,172.940,28.436,155.179
C07058=1067.288,156.605,421.871,172.939,28.433,155.179
C07059=1067.282,156.357,421.893,172.937,28.430,155.178
C07060=1067.276,156.107,421.914,172.934,28.427,155.178
C07061=1067.270,155.859,421.936,172.933,28.425,155.177
C07062=1067.265,155.609,421.958,172.931,28.421,155.177
C07063=1067.259,155.360,421.980,172.930,28.419,155.176
C07064=1067.253,155.112,422.001,172.927,28.416,155.176
C07065=1067.247,154.862,422.022,172.926,28.413,155.176
C07066=1067.241,154.614,422.044,172.924,28.410,155.175
C07067=1067.235,154.365,422.065,172.922,28.408,155.175
C07068=1067.230,154.116,422.087,172.920,28.405,155.174
C07069=1067.225,153.866,422.108,172.918,28.402,155.174
C07070=1067.219,153.618,422.129,172.917,28.399,155.174
C07071=1067.213,153.368,422.151,172.915,28.396,155.173
C07072=1067.207,153.119,422.173,172.914,28.394,155.173
C07073=1067.201,152.871,422.194,172.911,28.391,155.172
C07074=1067.195,152.621,422.216,172.909,28.388,155.172
C07075=1067.189,152.373,422.237,172.908,28.385,155.172
C07076=1067.184,152.123,422.258,172.906,28.382,155.171
C07077=1067.178,151.875,422.279,172.904,28.379,155.171
C07078=1067.172,151.625,422.301,172.902,28.377,155.170
C07079=1067.167,151.377,422.322,172.901,28.374,155.170
C07080=1067.161,151.127,422.343,172.899,28.371,155.170
C07081=1067.156,150.878,422.365,172.897,28.368,155.169
C07082=1067.149,150.629,422.386,172.895,28.365,155.169
C07083=1067.144,150.381,422.408,172.893,28.363,155.168
C07084=1067.138,150.131,422.429,172.892,28.360,155.168
C07085=1067.132,149.882,422.450,172.890,28.357,155.168
C07086=1067.126,149.633,422.471,172.888,28.354,155.167
C07087=1067.121,149.384,422.493,172.886,28.352,155.167
C07088=1067.115,149.135,422.514,172.884,28.349,155.166
C07089=1067.109,148.886,422.535,172.883,28.346,155.166
C07090=1067.104,148.638,422.556,172.881,28.343,155.166
C07091=1067.098,148.388,422.577,172.879,28.340,155.165
C07092=1067.092,148.139,422.598,172.877,28.338,155.165
C07093=1067.086,147.890,422.620,172.876,28.335,155.164
C07094=1067.081,147.641,422.641,172.874,28.332,155.164
C07095=1067.075,147.392,422.662,172.872,28.329,155.164
C07096=1067.070,147.143,422.683,172.870,28.326,155.163
C07097=1067.063,146.894,422.704,172.868,28.324,155.163
C07098=1067.057,146.645,422.725,172.867,28.321,155.162
C07099=1067.051,146.395,422.746,172.865,28.318,155.162
C07100=1067.046,146.147,422.767,172.864,28.315,155.162
C07101=1067.040,145.897,422.788,172.861,28.313,155.161
C07102=1067.034,145.649,422.809,172.859,28.310,155.161
C07103=1067.029,145.399,422.830,172.858,28.307,155.161
C07104=1067.022,145.151,422.851,172.856,28.305,155.160
C07105=1067.017,144.901,422.872,172.855,28.302,155.160
C07106=1067.011,144.652,422.893,172.853,28.299,155.159
C07107=1067.005,144.403,422.914,172.851,28.296,155.159
C07108=1066.999,144.154,422.935,172.849,28.293,155.159
C07109=1066.994,143.905,422.956,172.847,28.291,155.158
C07110=1066.988,143.656,422.977,172.846,28.288,155.158
C07111=1066.982,143.407,422.998,172.844,28.285,155.157
C07112=1066.975,143.124,423.022,172.842,28.282,155.157
C07113=1066.969,142.841,423.046,172.840,28.279,155.156
C07114=1066.963,142.557,423.070,172.838,28.275,155.156
C07115=1066.956,142.274,423.093,172.836,28.273,155.156
C07116=1066.950,142.025,423.114,172.835,28.270,155.155
C07117=1066.944,141.775,423.135,172.833,28.267,155.155
C07118=1066.939,141.526,423.155,172.831,28.264,155.154
C07119=1066.933,141.278,423.177,172.829,28.261,155.154
C07120=1066.928,141.028,423.197,172.827,28.259,155.154
C07121=1066.921,140.780,423.218,172.826,28.256,155.153
C07122=1066.916,140.531,423.239,172.824,28.253,155.153
C07123=1066.910,140.281,423.260,172.823,28.250,155.152
C07124=1066.905,140.032,423.281,172.820,28.247,155.152
C07125=1066.898,139.783,423.301,172.819,28.245,155.152
C07126=1066.893,139.534,423.322,172.817,28.242,155.151
C07127=1066.887,139.285,423.343,172.815,28.239,155.151
C07128=1066.881,139.036,423.363,172.814,28.236,155.150
C07129=1066.875,138.786,423.384,172.812,28.234,155.150
C07130=1066.870,138.537,423.404,172.811,28.231,155.149
C07131=1066.863,138.288,423.426,172.808,28.228,155.149
C07132=1066.858,138.039,423.446,172.807,28.225,155.149
C07133=1066.853,137.790,423.467,172.805,28.222,155.148
C07134=1066.847,137.541,423.487,172.803,28.220,155.148
C07135=1066.841,137.292,423.508,172.802,28.217,155.147
C07136=1066.835,137.043,423.528,172.800,28.214,155.147
C07137=1066.829,136.794,423.549,172.799,28.211,155.147
C07138=1066.823,136.544,423.570,172.796,28.209,155.146
C07139=1066.817,136.296,423.590,172.795,28.206,155.146
C07140=1066.812,136.047,423.611,172.793,28.203,155.146
C07141=1066.805,135.798,423.631,172.791,28.201,155.145
C07142=1066.800,135.548,423.652,172.790,28.198,155.145
C07143=1066.795,135.299,423.672,172.788,28.195,155.144
C07144=1066.789,135.051,423.692,172.787,28.192,155.144
C07145=1066.783,134.801,423.714,172.785,28.190,155.144
C07146=1066.777,134.552,423.734,172.783,28.187,155.143
C07147=1066.771,134.303,423.754,172.781,28.184,155.143
C07148=1066.765,134.054,423.775,172.780,28.181,155.142
C07149=1066.760,133.805,423.795,172.778,28.178,155.142
C07150=1066.754,133.556,423.815,172.776,28.176,155.142
C07151=1066.748,133.307,423.836,172.775,28.173,155.141
C07152=1066.743,133.058,423.856,172.773,28.170,155.141
C07153=1066.736,132.808,423.877,172.772,28.167,155.140
C07154=1066.731,132.559,423.897,172.769,28.164,155.140
C07155=1066.725,132.310,423.917,172.768,28.162,155.140
C07156=1066.720,132.062,423.938,172.766,28.159,155.139
C07157=1066.713,131.812,423.959,172.764,28.156,155.139
C07158=1066.708,131.563,423.979,172.763,28.153,155.138
C07159=1066.702,131.314,423.999,172.761,28.151,155.138
C07160=1066.696,131.065,424.019,172.760,28.148,155.138
C07161=1066.689,130.816,424.040,172.758,28.146,155.137
C07162=1066.684,130.566,424.059,172.757,28.143,155.137
C07163=1066.678,130.317,424.079,172.754,28.140,155.136
C07164=1066.672,130.068,424.100,172.752,28.137,155.136
C07165=1066.666,129.819,424.120,172.751,28.134,155.136
C07166=1066.660,129.570,424.140,172.749,28.132,155.135
C07167=1066.654,129.321,424.160,172.748,28.129,155.135
C07168=1066.649,129.072,424.181,172.746,28.127,155.135
C07169=1066.643,128.822,424.201,172.745,28.124,155.134
C07170=1066.637,128.574,424.221,172.743,28.121,155.134
C07171=1066.631,128.325,424.241,172.741,28.118,155.133
C07172=1066.625,128.076,424.262,172.740,28.116,155.133
C07173=1066.619,127.826,424.282,172.737,28.113,155.133
C07174=1066.613,127.577,424.301,172.736,28.110,155.132
C07175=1066.607,127.328,424.321,172.734,28.108,155.132
C07176=1066.601,127.045,424.345,172.733,28.104,155.131
C07177=1066.594,126.761,424.367,172.730,28.101,155.131
C07178=1066.587,126.478,424.390,172.729,28.098,155.130
C07179=1066.580,126.194,424.413,172.727,28.095,155.130
C07180=1066.574,125.945,424.433,172.726,28.092,155.130
C07181=1066.569,125.696,424.453,172.724,28.090,155.129
C07182=1066.563,125.447,424.473,172.722,28.087,155.129
C07183=1066.557,125.198,424.493,172.720,28.084,155.128
C07184=1066.551,124.949,424.512,172.718,28.082,155.128
C07185=1066.546,124.699,424.533,172.717,28.079,155.128
C07186=1066.540,124.450,424.553,172.715,28.076,155.127
C07187=1066.534,124.201,424.573,172.714,28.073,155.127
C07188=1066.528,123.952,424.593,172.712,28.071,155.127
C07189=1066.523,123.703,424.613,172.711,28.068,155.126
C07190=1066.517,123.454,424.633,172.709,28.065,155.126
C07191=1066.511,123.205,424.653,172.707,28.062,155.125
C07192=1066.505,122.956,424.672,172.706,28.060,155.125
C07193=1066.499,122.707,424.692,172.704,28.057,155.125
C07194=1066.493,122.457,424.713,172.703,28.054,155.124
C07195=1066.487,122.207,424.732,172.701,28.051,155.124
C07196=1066.481,121.959,424.752,172.699,28.048,155.123
C07197=1066.475,121.710,424.772,172.697,28.045,155.123
C07198=1066.470,121.460,424.792,172.696,28.043,155.123
C07199=1066.464,121.211,424.812,172.694,28.040,155.122
C07200=1066.458,120.962,424.832,172.692,28.038,155.122
C07201=1066.453,120.713,424.851,172.691,28.035,155.121
C07202=1066.447,120.464,424.871,172.689,28.032,155.121
C07203=1066.441,120.215,424.890,172.688,28.029,155.121
C07204=1066.436,119.966,424.911,172.686,28.027,155.120
C07205=1066.430,119.717,424.931,172.685,28.024,155.120
C07206=1066.424,119.467,424.950,172.683,28.021,155.119
C07207=1066.418,119.219,424.970,172.682,28.018,155.119
C07208=1066.413,118.969,424.989,172.680,28.016,155.119
C07209=1066.407,118.720,425.010,172.678,28.013,155.118
C07210=1066.401,118.471,425.030,172.677,28.010,155.118
C07211=1066.396,118.222,425.049,172.675,28.007,155.117
C07212=1066.390,117.973,425.069,172.674,28.004,155.117
C07213=1066.384,117.724,425.088,172.672,28.002,155.117
C07214=1066.378,117.475,425.108,172.671,27.999,155.116
C07215=1066.373,117.225,425.128,172.669,27.996,155.116
C07216=1066.367,116.976,425.148,172.667,27.993,155.115
C07217=1066.361,116.727,425.167,172.665,27.990,155.115
C07218=1066.355,116.478,425.187,172.664,27.988,155.115
C07219=1066.350,116.228,425.207,172.662,27.985,155.114
C07220=1066.344,115.980,425.227,172.660,27.982,155.114
C07221=1066.338,115.730,425.246,172.659,27.979,155.113
C07222=1066.333,115.480,425.266,172.657,27.976,155.113
C07223=1066.327,115.232,425.286,172.656,27.974,155.113
C07224=1066.321,114.982,425.305,172.654,27.971,155.112
C07225=1066.315,114.733,425.325,172.653,27.968,155.112
C07226=1066.310,114.484,425.344,172.651,27.965,155.111
C07227=1066.304,114.235,425.364,172.650,27.963,155.111
C07228=1066.298,113.986,425.383,172.648,27.960,155.111
C07229=1066.292,113.736,425.402,172.647,27.957,155.110
C07230=1066.286,113.488,425.422,172.645,27.954,155.110
C07231=1066.281,113.238,425.442,172.643,27.952,155.109
C07232=1066.275,112.989,425.461,172.642,27.949,155.109
C07233=1066.269,112.740,425.481,172.640,27.946,155.109
C07234=1066.263,112.490,425.500,172.639,27.943,155.108
C07235=1066.257,112.241,425.519,172.637,27.940,155.108
C07236=1066.251,111.992,425.539,172.636,27.938,155.107
C07237=1066.246,111.743,425.559,172.634,27.935,155.107
C07238=1066.239,111.494,425.577,172.633,27.933,155.107
C07239=1066.233,111.245,425.597,172.631,27.930,155.106
C07240=1066.228,110.961,425.618,172.630,27.927,155.106
C07241=1066.221,110.678,425.641,172.627,27.924,155.105
C07242=1066.214,110.394,425.662,172.626,27.921,155.105
C07243=1066.207,110.111,425.685,172.624,27.917,155.104
C07244=1066.202,109.861,425.704,172.623,27.915,155.104
C07245=1066.195,109.612,425.723,172.621,27.912,155.104
C07246=1066.189,109.363,425.743,172.619,27.910,155.103
C07247=1066.184,109.114,425.762,172.618,27.907,155.103
C07248=1066.178,108.864,425.781,172.616,27.904,155.103
C07249=1066.172,108.615,425.800,172.615,27.901,155.102
C07250=1066.166,108.366,425.819,172.613,27.898,155.102
C07251=1066.160,108.117,425.839,172.612,27.896,155.101
C07252=1066.154,107.868,425.858,172.609,27.893,155.101
C07253=1066.148,107.618,425.877,172.608,27.890,155.101
C07254=1066.143,107.370,425.896,172.606,27.887,155.100
C07255=1066.137,107.120,425.915,172.604,27.885,155.100
C07256=1066.131,106.871,425.934,172.603,27.882,155.100
C07257=1066.125,106.621,425.953,172.601,27.879,155.099
C07258=1066.119,106.373,425.973,172.600,27.877,155.099
C07259=1066.113,106.123,425.992,172.598,27.874,155.098
C07260=1066.107,105.874,426.011,172.597,27.871,155.098
C07261=1066.102,105.625,426.031,172.595,27.868,155.098
C07262=1066.096,105.376,426.049,172.594,27.865,155.097
C07263=1066.090,105.127,426.068,172.592,27.863,155.097
C07264=1066.084,104.877,426.087,172.591,27.860,155.096
C07265=1066.078,104.628,426.106,172.589,27.857,155.096
C07266=1066.072,104.379,426.125,172.588,27.854,155.095
C07267=1066.067,104.129,426.144,172.586,27.852,155.095
C07268=1066.061,103.880,426.164,172.584,27.849,155.095
C07269=1066.055,103.631,426.182,172.583,27.847,155.094
C07270=1066.049,103.382,426.201,172.581,27.844,155.094
C07271=1066.044,103.133,426.221,172.580,27.841,155.094
C07272=1066.037,102.883,426.239,172.579,27.838,155.093
C07273=1066.032,102.634,426.258,172.578,27.836,155.093
C07274=1066.027,102.385,426.277,172.576,27.833,155.092
C07275=1066.021,102.136,426.297,172.575,27.830,155.092
C07276=1066.014,101.887,426.315,172.573,27.827,155.092
